			E_MA_EVENT.MA_MOVE:
				M_SetMode(RefCtrl.nMode);	
				M_SetStatus('Moving  ...');
				IF (RefStat.nMode = MA_MODE_ENG) THEN
					// Set nCyclesIdle to zero.
					// Needed to distinguish if the motor is about to move off or it completed the move.
					RefStat.nSkippedCycles	:= 0;
					M_NextMove();		// Set new position and move absolute
					SetState(E_MA_STATE.OP, E_MA_SUBSTATE.OP_MOVING);
				ELSE
					M_NextMove();
//					SetState(E_MA_STATE.OP, E_MA_SUBSTATE.OP_TRACKING);
					SetState(E_MA_STATE.OP, E_MA_SUBSTATE.OP_PRESETTING);
				END_IF
			E_MA_EVENT.START_TRACK:
				M_SetMode(RefCtrl.nMode);	
				// Set nCyclesIdle to zero.
				// Needed to distinguish if the motor is about to move off or it completed the move.
				RefStat.nSkippedCycles 	:= 0;	// Delayed action
				M_NextMoveAbs();
//				SetState(E_MA_STATE.OP, E_MA_SUBSTATE.OP_TRACKING);
				SetState(E_MA_STATE.OP, E_MA_SUBSTATE.OP_PRESETTING);
			E_MA_EVENT.PRESETDONE:
				// Preset is done, start tracking.
				SetState(E_MA_STATE.OP, E_MA_SUBSTATE.OP_TRACKING);
			E_MA_EVENT.TRACKEXIT:
				// Tracking is not good, it's more like presetting.
				SetState(E_MA_STATE.OP, E_MA_SUBSTATE.OP_PRESETTING);
		END_CASE
END_CASE
END_METHOD

{attribute 'TcRpcEnable':='1'}
METHOD RPC_Init : INT
VAR_INPUT
END_VAR

VAR 
	i: INT;
	bMotorMoving:	BOOL := FALSE;
END_VAR
// Log similar string in every derived FB
//M_LogEventGeneral('Initialising MA motors');

//
// Check if it is safe to operate motors.
//
IF NOT in_bSafe	THEN
	RPC_Init	:= M_SetRpcStatus(E_MA_RPC_ERROR.UNSAFE);
	RETURN;
END_IF


// It does all the verifications for the MOTOR device before
// triggering the Init event.

FOR i := 1 TO nNumAxes DO
	// RPC calls are not allowed in Local mode.
	// Fail on the first occurrence.
	IF ptrMotorStat[i]^.bLocal THEN
		RPC_Init	:= M_SetRpcStatus(E_MA_RPC_ERROR.LOCAL);
		RETURN;
	END_IF

	// If any of the motors is moving, RPC_Init() will fail.
	// However, the moving motor will be stopped, so next INIT will be OK.
	// We loop through all motors.
	IF	ptrMotorStat[i]^.nState = E_MOTOR_STATE.OP	AND  
		ptrMotorStat[i]^.nSubstate <> E_MOTOR_SUBSTATE.OP_STANDSTILL	THEN
		// There is a moving motor in the system.
		bMotorMoving	:= TRUE;
		// Stop the motor.
		// Send STOP command to the motors.
		ptrMotorCtrl[i]^.nCommand	:= E_MOTOR_COMMAND.STOP;
		ptrMotorCtrl[i]^.bExecute	:= TRUE;
		// RPC_Init() will fail !!!
		RPC_Init	:= M_SetRpcStatus(E_MA_RPC_ERROR.INIT_WHILE_MOVING);
	END_IF
END_FOR

IF bMotorMoving THEN
	// RPC_Init is already set to failure.
	RETURN;
ELSE
	// Proceed with INIT.
	RefCtrl.nCommand := E_MA_COMMAND.INIT;
	RefCtrl.bExecute := TRUE;
		
	// Call was successful
	RPC_Init	:= M_SetRpcStatus(E_MA_RPC_ERROR.OK);
END_IF
END_METHOD

METHOD SetAction
VAR_INPUT
	actionName:		STRING;
END_VAR

RefStat.sm.sActionDesc := actionName;
END_METHOD

METHOD SetEvent
VAR_INPUT
	nEventId:			DINT;
END_VAR

nEvent := nEventId;

CASE nEventId OF
	E_MA_EVENT.NONE:
		RefStat.sm.sEventDesc := '';
		RETURN;
		
	E_MA_EVENT.RESET:
		RefStat.sm.sEventDesc := 'CMD RESET';
		RETURN;
	
	E_MA_EVENT.INIT:
		RefStat.sm.sEventDesc := 'CMD INIT';
		RETURN;

	E_MA_EVENT.STOP:
		RefStat.sm.sEventDesc := 'CMD STOP';
		RETURN;

	E_MA_EVENT.ENABLE:
		RefStat.sm.sEventDesc := 'CMD ENABLE';
		RETURN;

	E_MA_EVENT.DISABLE:
		RefStat.sm.sEventDesc := 'CMD DISABLE';
		RETURN;
		
	E_MA_EVENT.MA_MOVE:
		RefStat.sm.sEventDesc := 'CMD MOVE';
		RETURN;
		
	E_MA_EVENT.START_TRACK:
		RefStat.sm.sEventDesc := 'CMD START_TRACK -> PRESETTING';
		RETURN;

	E_MA_EVENT.STOP_TRACK:
		RefStat.sm.sEventDesc := 'CMD STOP_TRACK';
		RETURN;
		
	E_MA_EVENT.PRESETDONE:
		RefStat.sm.sEventDesc := 'TRACKING';
		RETURN;
		
	E_MA_EVENT.TRACKEXIT:
		RefStat.sm.sEventDesc := 'TRACKING -> PRESETTING';
		RETURN;
		
	E_MA_EVENT.HWOK:
		RefStat.sm.sEventDesc := 'SIG HWOK';
		RETURN;

	E_MA_EVENT.ERRHW:
		RefStat.sm.sEventDesc := 'INT ERRHW';
		RETURN;
	
	E_MA_EVENT.UNSAFE:
		RefStat.sm.sEventDesc := 'EXT UNSAFE';
		RETURN;
	
END_CASE 

(* INTERNAL ERROR *)
RefStat.sm.sEventDesc := 'UNKNOWN EVENT';
END_METHOD

// Set the state and substate of the device
METHOD SetState : BOOL
VAR_INPUT
	in_nState:		INT;
	in_nSubstate:	INT;
END_VAR

(* 
	Update State Machine active state configuration.
*)

IF in_nState <> E_MA_STATE.NONE THEN
	RefStat.sm.nState	:= in_nState;
END_IF
IF in_nSubstate <> E_MA_SUBSTATE.NONE THEN
	RefStat.sm.nSubstate	:= in_nSubstate;
END_IF

(* Update active state configuration description *)

IF in_nState = E_MA_STATE.NOTOP THEN
	RefStat.sm.sState	:= 'NOT OP';
ELSIF in_nState = E_MA_STATE.OP THEN
	RefStat.sm.sState	:= 'OPERATIONAL';
END_IF

IF in_nSubstate = E_MA_SUBSTATE.NOTOP_NOTREADY THEN
	RefStat.sm.sSubstate	:= 'NOT READY';
ELSIF in_nSubstate = E_MA_SUBSTATE.NOTOP_INITIALISING THEN
	RefStat.sm.sSubstate	:= 'INITIALISING';
ELSIF in_nSubstate = E_MA_SUBSTATE.NOTOP_READY THEN
	RefStat.sm.sSubstate	:= 'READY';
ELSIF in_nSubstate = E_MA_SUBSTATE.NOTOP_ERROR THEN
	RefStat.sm.sSubstate	:= 'ERROR';
ELSIF in_nSubstate = E_MA_SUBSTATE.OP_DISABLING THEN
	RefStat.sm.sSubstate	:= 'DISABLING';
ELSIF in_nSubstate = E_MA_SUBSTATE.OP_MOVING THEN
	RefStat.sm.sSubstate	:= 'MOVING';
ELSIF in_nSubstate = E_MA_SUBSTATE.OP_STANDSTILL THEN
	RefStat.sm.sSubstate	:= 'STANDSTILL';
ELSIF in_nSubstate = E_MA_SUBSTATE.OP_TRACKING THEN
	RefStat.sm.sSubstate	:= 'TRACKING';
ELSIF in_nSubstate = E_MA_SUBSTATE.OP_PRESETTING THEN
	RefStat.sm.sSubstate	:= 'PRESETTING';
ELSIF in_nSubstate = E_MA_SUBSTATE.OP_STOPPING THEN
	RefStat.sm.sSubstate	:= 'STOPPING';
ELSIF in_nSubstate = E_MA_SUBSTATE.OP_ERROR THEN
	RefStat.sm.sSubstate	:= 'ERROR';
ELSE
	RefStat.sm.sSubstate	:= '';
END_IF
END_METHOD

METHOD User_ComputeNextPos : BOOL
VAR_INPUT
END_VAR
VAR
	i:	int;
END_VAR
// TODOUSER: Calculate next position for each axes based on the current mode.
IF RefStat.nMode = MA_MODE_ENG THEN
	FOR i := 1 TO nNumAxes DO
		;
	END_FOR
END_IF
END_METHOD

// Method for hard-coding of configuration parameters by the User.
METHOD User_Configure : BOOL
VAR_INPUT
END_VAR
VAR
	i:	INT;
END_VAR
//
// TODOUSER: Configure anything that is different from default configuration or
//           that has to take all motors into account.
//

//
// This is mandatory.
//
// Set the global timeouts to the longest ones. 
FOR i := 1 TO nNumAxes DO
	IF ptrMotorCfg[i]^.nTimeoutInit > RefCfg.timeout.nInitTimeout THEN
		RefCfg.timeout.nInitTimeout  := ptrMotorCfg[i]^.nTimeoutInit;
	END_IF
	IF ptrMotorCfg[i]^.nTimeoutMove > RefCfg.timeout.nMoveTimeout THEN
		RefCfg.timeout.nMoveTimeout  := ptrMotorCfg[i]^.nTimeoutMove;
	END_IF
END_FOR

//
// TODOUSER: Any other configuration
//
END_METHOD

// User Method executed on each cycle before processing events and states.
METHOD User_GetParams : BOOL
VAR_INPUT
END_VAR
VAR
	i:	INT;
END_VAR
//
// TODOUSER: Set anything that should be set on every cycle, if any.
//

// Example: Any settings that are mode dependant.
CASE RefCtrl.nMode OF
			MA_MODE_ENG:
			    ; 
END_CASE
END_METHOD

// User Method executed on each cycle after processing events and states.
METHOD User_SetParams : BOOL
VAR_INPUT
END_VAR
VAR
	i:		INT;
END_VAR
//
// Mandatory
//
// Set maximum positioning error
RefStat.lrPosError	:= M_GetMaxPosError();


// TODO Add code for handling individual axes, if any.
FOR i := 1 TO nNumAxes DO
	;
END_FOR
END_METHOD

END_FUNCTION_BLOCK

// ---- POUs/MultiAxis/FB_MA_DROT.TcPOU
FUNCTION_BLOCK FB_MA_DROT EXTENDS FB_MA_BASE
VAR_INPUT
	{attribute 'OPC.UA.DA' := '0'}
	sMotorName:			STRING	:= 'Motor';	(* Default Motor name *)
	{attribute 'OPC.UA.DA' := '0'}
	in_lrRotation: LREAL := 0; (* Rotation used for Sky mode *)
	{attribute 'OPC.UA.DA' := '0'}
	in_lrPupil: LREAL := 0; (* Pupil rotation for Elevation mode *)
	{attribute 'OPC.UA.DA' := '0'}
	in_lrParallactic: LREAL := 0; (* Parallactic angle *)
	{attribute 'OPC.UA.DA' := '0'}
	nNOVRAM_DevId:	UDINT	:= 0;		(* NOVRAM device ID - normally 4 *)
	{attribute 'OPC.UA.DA' := '0'}
	nNOVRAM_Offset:	UDINT	:= 0;		(* NOVRAM offset where motor configuration is stored *)
END_VAR
VAR_OUTPUT
END_VAR
VAR

	
	{attribute 'OPC.UA.DA' := '1'}
	cfg:				T_DROT_CFG;
	{attribute 'OPC.UA.DA' := '1'}
	ctrl:				T_DROT_CTRL;
	{attribute 'OPC.UA.DA' := '1'}
	stat:				T_DROT_STAT;
	
	{attribute 'OPC.UA.DA':='1'}
	motor:              FB_MOTOR;
	
END_VAR


// A MUST !!! Set references to real structures
RefCfg		REF=cfg;
RefCtrl		REF=ctrl;
RefStat		REF=stat;


motor(	sName 				:= sMotorName,	
		in_bSafe			:= in_bSafe,
		in_bDisableIfUnsafe	:= in_bDisableIfUnsafe,
		nNOVRAM_DevId 		:= nNOVRAM_DevId, 
		nNOVRAM_Offset 		:= nNOVRAM_Offset);

SUPER^(nNumAxes:=1, pMotor1:=ADR(motor));

METHOD M_LogCommand : BOOL
VAR
	cmd:	INT;
	mode:	INT;
	sLog:	STRING;
END_VAR
cmd		:= RefCtrl.nCommand;
mode	:= ctrl.nMode;

// Log DROT command.
// Set motor logging to FALSE when tracking,
// in order to reduce flooding of logs.
IF cmd = E_MA_COMMAND.RESET THEN
	pMotor1^.RPC_SetLog(TRUE);
	M_SetStatus('Resetting DROT device...');		
	M_LogEventGeneral('Resetting DROT device...');
ELSIF cmd = E_MA_COMMAND.ENABLE THEN
	pMotor1^.RPC_SetLog(TRUE);
	M_SetStatus('');		
	M_LogEventGeneral('Enabling DROT device...');
ELSIF cmd = E_MA_COMMAND.INIT THEN
	pMotor1^.RPC_SetLog(TRUE);
	M_SetStatus('Initialising DROT device...');		
	M_LogEventGeneral('Initialising DROT device...');
ELSIF cmd = E_MA_COMMAND.START_TRACK THEN
	pMotor1^.RPC_SetLog(FALSE);
	IF mode= E_DROT_MODE.ELEV THEN
		M_SetStatus('Tracking in ELEV mode');
		sLog	:= LREAL_TO_STRING(ctrl.lrPosang);
		sLog	:= CONCAT('Setting DROT to ELEVATION mode. Angle = ', sLog);
		M_LogEventGeneral(sLog);
	ELSIF mode= E_DROT_MODE.SKY THEN
		M_SetStatus('Tracking in SKY mode');
		sLog	:= LREAL_TO_STRING(ctrl.lrPosang);
		sLog	:= CONCAT('Setting DROT to SKY mode. Angle = ', sLog);
		M_LogEventGeneral(sLog);
	ELSIF mode= E_DROT_MODE.USER THEN
		M_SetStatus('Tracking in USER mode');
		sLog	:= LREAL_TO_STRING(ctrl.lrPosang);
		sLog	:= CONCAT('Setting DROT to USER mode. Angle = ', sLog);
		M_LogEventGeneral(sLog);
	END_IF
ELSIF cmd = E_MA_COMMAND.DISABLE THEN
	M_SetStatus('');		
	M_LogEventGeneral('Disabling DROT device...');
ELSIF cmd = E_MA_COMMAND.STOP THEN
	pMotor1^.RPC_SetLog(TRUE);
	M_LogEventGeneral('Stopping DROT device...');
ELSIF cmd = E_MA_COMMAND.STOP_TRACK THEN
	pMotor1^.RPC_SetLog(TRUE);
	IF mode= E_DROT_MODE.ENG THEN
		M_SetStatus('Moving to Engineering position ...');		
		sLog	:= LREAL_TO_STRING(stat.lrPos);
		sLog	:= CONCAT('Setting DROT to ENG mode. Angle = ', sLog);
		M_LogEventGeneral(sLog);
	ELSIF mode= E_DROT_MODE.STAT THEN
		M_SetStatus('Moving to STAT position ...');		
		sLog	:= LREAL_TO_STRING(stat.lrPos);
		sLog	:= CONCAT('Setting DROT to STAT mode. Angle = ', sLog);
		M_LogEventGeneral(sLog);
	END_IF
END_IF
END_METHOD

{attribute 'TcRpcEnable':='1'}
METHOD RPC_Disable : INT
VAR_INPUT
END_VAR

// It does all the verifications for the MOTOR device before
// triggering the Init event.

// RPC calls are not allowed in Local mode.
IF ptrMotorStat[1]^.bLocal THEN
	RPC_Disable	:= M_SetRpcStatus(E_MA_RPC_ERROR.LOCAL);
	RETURN;
END_IF

// Disable command is accepted only if device is in OP state.
IF ptrMotorStat[1]^.nState <> E_MOTOR_STATE.OP THEN
	RPC_Disable	:= M_SetRpcStatus(E_MA_RPC_ERROR.NOT_OP);
	RETURN;
ELSE
	// Set disable command
	RefCtrl.nCommand := E_MA_COMMAND.DISABLE;
	RefCtrl.bExecute := TRUE;
	
	// Call was successful
	RPC_Disable	:= M_SetRpcStatus(E_MA_RPC_ERROR.OK);
END_IF
END_METHOD

{attribute 'TcRpcEnable':='1'}
METHOD RPC_Enable : INT
VAR_INPUT
END_VAR

// It does all the verifications for the MOTOR device before
// triggering the Enable event.

//
// Check if it is safe to operate motors.
//
IF NOT in_bSafe	THEN
	RPC_Enable	:= M_SetRpcStatus(E_MA_RPC_ERROR.UNSAFE);
	RETURN;
END_IF



// RPC calls are not allowed in Local mode.
IF ptrMotorStat[1]^.bLocal THEN
	RPC_Enable	:= M_SetRpcStatus(E_MA_RPC_ERROR.LOCAL);
	RETURN;
END_IF

// Enable command is accepted only if device is in NOTOP_READY.
IF	ptrMotorStat[1]^.nSubstate <> E_MOTOR_SUBSTATE.NOTOP_READY		THEN
	RPC_Enable	:= M_SetRpcStatus(E_MA_RPC_ERROR.NOT_NOTOP_READY);
	RETURN;
ELSE
	// Set enable command
	RefCtrl.nCommand := E_MA_COMMAND.ENABLE;
	RefCtrl.bExecute := TRUE;
	
	// Call was successful
	RPC_Enable	:= M_SetRpcStatus(E_MA_RPC_ERROR.OK);
END_IF
END_METHOD

{attribute 'TcRpcEnable':='1'}
METHOD RPC_Init : INT
VAR_INPUT
END_VAR

VAR
END_VAR
M_LogEventGeneral('Initialising DROT motor...');

//
// Check if it is safe to operate motors.
//
IF NOT in_bSafe	THEN
	RPC_Init	:= M_SetRpcStatus(E_MA_RPC_ERROR.UNSAFE);
	RETURN;
END_IF


RPC_Init	:= SUPER^.RPC_Init();
END_METHOD

{attribute 'TcRpcEnable':='1'}
METHOD RPC_MoveAbs : INT
VAR_INPUT
	in_lrPos:	LREAL;
	in_lrVel:	LREAL;
END_VAR
//
// Check if it is safe to operate motors.
//
IF NOT in_bSafe	THEN
	RPC_MoveAbs	:= M_SetRpcStatus(E_MA_RPC_ERROR.UNSAFE);
	RETURN;
END_IF


// RPC calls are not allowed in Local mode.
IF motor.stat.bLocal THEN
	RPC_MoveAbs	:= M_SetRpcStatus(E_MA_RPC_ERROR.LOCAL);
	RETURN;
// Move Absolute command is accepted only in OP state.
ELSIF	motor.stat.nState <> E_MOTOR_STATE.OP	THEN
	RPC_MoveAbs	:= M_SetRpcStatus(E_MA_RPC_ERROR.NOT_OP);
	RETURN;
ELSIF	stat.sm.nState <> E_MA_STATE.OP	THEN
	RPC_MoveAbs	:= M_SetRpcStatus(E_MA_RPC_ERROR.NOT_OP);
	RETURN;
// Set velocity cannot be <=0.0.
ELSIF	in_lrVel <= 0.0	THEN
	RPC_MoveAbs	:= M_SetRpcStatus(E_MOTOR_RPC_ERROR.VEL_NEG);
	RETURN;
// Set velocity cannot be greater than MAX Velocity.
ELSIF	in_lrVel > motor.stat.axis.lrMaxVelocity	THEN
	RPC_MoveAbs	:= M_SetRpcStatus(E_MOTOR_RPC_ERROR.VEL_MAX);
	RETURN;
END_IF


SetState(E_MA_STATE.OP, E_MA_SUBSTATE.OP_MOVING);
// Set command
ctrl.nCommand 		:= E_MA_COMMAND.MA_MOVE;
ctrl.nMode          := E_DROT_MODE.ENG;
ctrl.lrTargetPos    := in_lrPos;
ctrl.lrTargetVel    := in_lrVel;
ctrl.bExecute 		:= TRUE;

// Call was successful
RPC_MoveAbs	:= M_SetRpcStatus(E_MA_RPC_ERROR.OK);
END_METHOD

{attribute 'TcRpcEnable':='1'}
METHOD RPC_MoveAngle : INT
VAR_INPUT
	in_lrAngle:	LREAL;
END_VAR
//
// Check if it is safe to operate motors.
//
IF NOT in_bSafe	THEN
	RPC_MoveAngle	:= M_SetRpcStatus(E_MA_RPC_ERROR.UNSAFE);
	RETURN;
END_IF



// RPC calls are not allowed in Local mode.
IF motor.stat.bLocal THEN
	RPC_MoveAngle	:= M_SetRpcStatus(E_MA_RPC_ERROR.LOCAL);
	RETURN;
// Move Absolute command is accepted only in OP state.
ELSIF	motor.stat.nState <> E_MOTOR_STATE.OP	THEN
	RPC_MoveAngle	:= M_SetRpcStatus(E_MA_RPC_ERROR.NOT_OP);
	RETURN;
ELSIF	stat.sm.nState <> E_MA_STATE.OP	THEN
	RPC_MoveAngle	:= M_SetRpcStatus(E_MA_RPC_ERROR.NOT_OP);
	RETURN;
END_IF


SetState(E_MA_STATE.OP, E_MA_SUBSTATE.OP_MOVING);
// Set command
ctrl.lrPosang 	:= in_lrAngle;
ctrl.nMode		:= E_DROT_MODE.STAT;
ctrl.nCommand	:= E_MA_COMMAND.STOP_TRACK;
ctrl.bExecute	:= TRUE;

// Call was successful
RPC_MoveAngle	:= M_SetRpcStatus(E_MA_RPC_ERROR.OK);
END_METHOD

{attribute 'TcRpcEnable':='1'}
METHOD RPC_MoveRel : INT
VAR_INPUT
	in_lrPos:	LREAL;
	in_lrVel:	LREAL;
END_VAR
//
// Check if it is safe to operate motors.
//
IF NOT in_bSafe	THEN
	RPC_MoveRel	:= M_SetRpcStatus(E_MA_RPC_ERROR.UNSAFE);
	RETURN;
END_IF


// RPC calls are not allowed in Local mode.
IF motor.stat.bLocal THEN
	RPC_MoveRel	:= M_SetRpcStatus(E_MA_RPC_ERROR.LOCAL);
	RETURN;
// Move Absolute command is accepted only in OP state.
ELSIF	motor.stat.nState <> E_MOTOR_STATE.OP	THEN
	RPC_MoveRel	:= M_SetRpcStatus(E_MA_RPC_ERROR.NOT_OP);
	RETURN;
ELSIF	stat.sm.nState <> E_MA_STATE.OP	THEN
	RPC_MoveRel	:= M_SetRpcStatus(E_MA_RPC_ERROR.NOT_OP);
	RETURN;
// Set velocity cannot be <=0.0.
ELSIF	in_lrVel <= 0.0	THEN
	RPC_MoveRel	:= M_SetRpcStatus(E_MOTOR_RPC_ERROR.VEL_NEG);
	RETURN;
// Set velocity cannot be greater than MAX Velocity.
ELSIF	in_lrVel > motor.stat.axis.lrMaxVelocity	THEN
	RPC_MoveRel	:= M_SetRpcStatus(E_MOTOR_RPC_ERROR.VEL_MAX);
	RETURN;
END_IF


SetState(E_MA_STATE.OP, E_MA_SUBSTATE.OP_MOVING);
// Set command
ctrl.nCommand 		:= E_MA_COMMAND.MA_MOVE;
ctrl.nMode          := E_DROT_MODE.ENG;
ctrl.lrTargetPos    := motor.stat.lrPosActual + in_lrPos;
ctrl.lrTargetVel    := in_lrVel;
ctrl.bExecute 		:= TRUE;

// Call was successful
RPC_MoveRel	:= M_SetRpcStatus(E_MA_RPC_ERROR.OK);
END_METHOD

{attribute 'TcRpcEnable':='1'}
METHOD RPC_MoveVel : INT
VAR_INPUT
	in_lrVel:	LREAL;
END_VAR
VAR
	dir:	DINT;
END_VAR
//
// Check if it is safe to operate motors.
//
IF NOT in_bSafe	THEN
	RPC_MoveVel	:= M_SetRpcStatus(E_MA_RPC_ERROR.UNSAFE);
	RETURN;
END_IF


IF	stat.sm.nState <> E_MA_STATE.OP	THEN
	RPC_MoveVel	:= M_SetRpcStatus(E_MA_RPC_ERROR.NOT_OP);
	RETURN;
ELSIF	in_lrVel = 0.0	THEN
// Set velocity cannot be 0.0.
	RPC_MoveVel	:= M_SetRpcStatus(E_MOTOR_RPC_ERROR.VEL_ZERO);
	RETURN;
END_IF

// Check velocity against Vel_max.
// Note: Negative velocity is accepted.
// Check if Velocity is too high.
IF ABS(in_lrVel) > ptrMotorStat[1]^.axis.lrMaxVelocity THEN
	RPC_MoveVel	:= M_SetRpcStatus(E_MOTOR_RPC_ERROR.VEL_MAX);
	RETURN;
END_IF


// Update State and Status
SetState(E_MA_STATE.OP, E_MA_SUBSTATE.OP_MOVING);
M_SetStatus('Moving in Velocity mode...');
ctrl.nMode	:= E_ADC_MODE.ENG;

// Set the direction of movement.
IF in_lrVel > 0.0	THEN
	dir	:= MC_Positive_Direction;
ELSE
	dir	:= MC_Negative_Direction;
END_IF

// This will command all the motors and restart the timer.
ActionMoveVelExecute(vel:=ABS(in_lrVel), dir:=dir);

// Call was successful
RPC_MoveVel	:= M_SetRpcStatus(E_MA_RPC_ERROR.OK);
END_METHOD

{attribute 'TcRpcEnable':='1'}
METHOD RPC_Reset : INT
VAR_INPUT
END_VAR

// RPC calls are not allowed in Local mode.
IF ptrMotorStat[1]^.bLocal THEN
	RPC_Reset	:= M_SetRpcStatus(E_MA_RPC_ERROR.LOCAL);
	RETURN;
END_IF

ctrl.nCommand := E_MA_COMMAND.RESET;
ctrl.bExecute := TRUE;

// Call was successful
RPC_Reset	:= M_SetRpcStatus(E_MA_RPC_ERROR.OK);
END_METHOD

{attribute 'TcRpcEnable':='1'}
METHOD RPC_StartTrack : INT
VAR_INPUT
	in_mode:	 INT := 2;
	in_angle:    LREAL := 0.0;
END_VAR
//
// Check if it is safe to operate motors.
//
IF NOT in_bSafe	THEN
	RPC_StartTrack	:= M_SetRpcStatus(E_MA_RPC_ERROR.UNSAFE);
	RETURN;
END_IF



// RPC calls are not allowed in Local mode.
IF ptrMotorStat[1]^.bLocal THEN
	RPC_StartTrack	:= M_SetRpcStatus(E_MA_RPC_ERROR.LOCAL);
	RETURN;
// Move Absolute command is accepted only in OP state.
ELSIF	ptrMotorStat[1]^.nState <> E_MOTOR_STATE.OP	THEN
	RPC_StartTrack	:= M_SetRpcStatus(E_MA_RPC_ERROR.NOT_OP);
	RETURN;
END_IF

// Set command
ctrl.lrPosang := in_angle;
ctrl.nMode:= in_mode;
ctrl.nCommand:=E_MA_COMMAND.START_TRACK;
ctrl.lrOffset := 0.0;
stat.lrTotalOffset := 0.0;
ctrl.bExecute:=(TRUE);

// Call was successful
RPC_StartTrack	:= M_SetRpcStatus(E_MA_RPC_ERROR.OK);
END_METHOD

{attribute 'TcRpcEnable':='1'}
METHOD RPC_Stop : INT
VAR_INPUT
END_VAR

// RPC calls are not allowed in Local mode.
IF ptrMotorStat[1]^.bLocal THEN
	RPC_Stop	:= M_SetRpcStatus(E_MA_RPC_ERROR.LOCAL);
	RETURN;
END_IF

ctrl.nCommand := E_MA_COMMAND.STOP;
ctrl.bExecute := TRUE;

RPC_Stop	:= M_SetRpcStatus(E_MA_RPC_ERROR.OK);
END_METHOD

{attribute 'TcRpcEnable':='1'}
METHOD RPC_StopTrack : INT
VAR_INPUT
END_VAR
VAR
	sLog:	STRING;
END_VAR
IF (RefStat.nMode >= E_DROT_MODE.SKY) THEN
	// RPC calls are not allowed in Local mode.
	IF ptrMotorStat[1]^.bLocal THEN
		RPC_StopTrack	:= M_SetRpcStatus(E_MA_RPC_ERROR.LOCAL);
		RETURN;
	END_IF

	sLog	:= LREAL_TO_STRING(stat.lrPos);
	sLog	:= CONCAT('Stopping Tracking. Angle = ', sLog);
	M_LogEventGeneral(sLog);

	RefCtrl.nMode           :=  E_DROT_MODE.STAT;
	// Set command
	RefCtrl.nCommand 		:= E_MA_COMMAND.STOP_TRACK;
	RefCtrl.bExecute 		:= TRUE;
END_IF

// Call was successful
RPC_StopTrack	:= M_SetRpcStatus(E_MA_RPC_ERROR.OK);
END_METHOD

{attribute 'TcRpcEnable':='1'}
METHOD RPC_TrackOffset : INT
VAR_INPUT
	in_lrOffset:	LREAL;
END_VAR
//
// Check if it is safe to operate motors.
//
IF NOT in_bSafe	THEN
	RPC_TrackOffset	:= M_SetRpcStatus(E_MA_RPC_ERROR.UNSAFE);
	RETURN;
END_IF


// RPC calls are not allowed in Local mode.
IF motor.stat.bLocal THEN
	RPC_TrackOffset	:= M_SetRpcStatus(E_MA_RPC_ERROR.LOCAL);
	RETURN;
// Move Absolute command is accepted only in OP state.
ELSIF	motor.stat.nState <> E_MOTOR_STATE.OP	THEN
	RPC_TrackOffset	:= M_SetRpcStatus(E_MA_RPC_ERROR.NOT_OP);
	RETURN;
ELSIF	(stat.nMode <= E_DROT_MODE.STAT) THEN
	RPC_TrackOffset	:= M_SetRpcStatus(E_MA_RPC_ERROR.NOT_TRACKING);
	RETURN;
END_IF

// Update offset
ctrl.lrOffset    := in_lrOffset;

// Call was successful
RPC_TrackOffset	:= M_SetRpcStatus(E_MA_RPC_ERROR.OK);
END_METHOD

METHOD User_ComputeNextPos : BOOL
VAR_INPUT
END_VAR
VAR
	fieldRotation: LREAL;
	modeAngle:     LREAL;
	pos:           LREAL := 0.0 ;
	posang:        LREAL;
END_VAR
// Handle various derotator modes
CASE RefCtrl.nMode OF
			E_DROT_MODE.STAT:
			    pos := cfg.lrStatRef + cfg.nDirSign * (ctrl.lrPosang)/2.0;
				stat.lrAngleOnSky := 0.0;
				stat.lrModeAngle := pos;
				ptrMotorCtrl[1]^.lrVelocity := ptrMotorCfg[1]^.lrDefaultVelocity;
			E_DROT_MODE.SKY:
				stat.lrTotalOffset := stat.lrTotalOffset + ctrl.lrOffset;
				ctrl.lrOffset := 0.0;
				fieldRotation := ctrl.lrRotation;
				pos := cfg.lrSkyRef + (cfg.nDirSign * ((ctrl.lrPosang - fieldRotation)/2)) + stat.lrTotalOffset ;
				stat.lrAngleOnSky := ctrl.lrPosang;
				stat.lrModeAngle := stat.lrAngleOnSky;
				ptrMotorCtrl[1]^.lrVelocity := ptrMotorCfg[1]^.lrDefaultVelocity;
			E_DROT_MODE.ELEV:
				stat.lrTotalOffset := stat.lrTotalOffset + ctrl.lrOffset;
				ctrl.lrOffset := 0.0;
				pos := cfg.lrElevRef + ((cfg.nFocusSign * cfg.nDirSign * (ctrl.lrPupil)) /2.0) + stat.lrTotalOffset;
				stat.lrAngleOnSky := ctrl.lrParallactic;
				stat.lrModeAngle := stat.lrAngleOnSky;
				ptrMotorCtrl[1]^.lrVelocity := ptrMotorCfg[1]^.lrDefaultVelocity;
			E_DROT_MODE.USER:
				//modeAngle := (parUser[1] * ctrl.lrPosang +
				//	          parUser[2] * i_trk_data.alt_deg +
				//			  parUser[3] * i_trk_data.pa_deg );
				//pos := cfg.lrUserRef + cfg.nDirSign * modeAngle;
				//stat.lrAngleOnSky := 0.0;
				//stat.lrModeAngle  := modeAngle;
			E_DROT_MODE.ENG:
				pos := ctrl.lrTargetPos;
		        ptrMotorCtrl[1]^.lrVelocity := ctrl.lrTargetVel;		
		        M_SetStatus('Moving to Engineering position ...');
END_CASE

// assign new TARGET position
ptrMotorCtrl[1]^.lrPosition := pos;
stat.lrPos := pos;	// Used in the DROT GUI as 'Target'
END_METHOD

// Method for hard-coding of configuration parameters by the User.
METHOD User_Configure : BOOL
VAR_INPUT
END_VAR
VAR
	i:	INT;
END_VAR
SUPER^.User_Configure();	// Mandatory!

//
// TODOUSER: Configure anything that is different from default configuration.
//
// Examples:
//

//
// Individual Motor configuration
ptrMotorCfg[1]^.nAxisType	        := E_MOTOR_AXIS_TYPE.CIRCULAR_OPTIMISED;
ptrMotorCfg[1]^.lrDefaultVelocity	:= 3.0;	// Set default velocity to 10 deg/sec


// Multi-axis system configuration
ctrl.lrPosang	    :=  0.0;	// Position angle for OFF mode, i.e. HOME position
ctrl.lrTargetPos	:=  0.0;	
ctrl.lrTargetVel	:= 3.0;	// Velocity for ENG mode
END_METHOD

// User Method executed on each cycle before processing events and states.
METHOD User_GetParams : BOOL
VAR_INPUT
END_VAR
VAR
	i:	INT;
END_VAR


SUPER^.User_GetParams();
END_METHOD

// User Method executed on each cycle after processing events and states.
METHOD User_SetParams : BOOL
VAR_INPUT
END_VAR
VAR
	i:		INT;
END_VAR
//
// Mandatory
//
SUPER^.User_SetParams();

// Set maximum positioning error
stat.lrPosError		:= M_GetMaxPosError();

// Check if we are tracking or still presetting.
// Tracking is OK if the positioning error is less than the threshold (bTrackingOK).
// Once device is tracking, it should go back to presetting if the error is greater
// than twice the threshold  (bTrackingBAD).
IF	ctrl.nMode = E_DROT_MODE.ELEV OR  
	ctrl.nMode = E_DROT_MODE.SKY  OR  
	ctrl.nMode = E_DROT_MODE.USER	THEN
	stat.bTrackingOK	:= SEL (stat.lrPosError <= cfg.lrTrkThreshold, FALSE, TRUE);
	stat.bTrackingBAD	:= SEL (stat.lrPosError > 2.0 * cfg.lrTrkThreshold, FALSE, TRUE);
	ctrl.lrRotation := in_lrRotation;
	ctrl.lrPupil := in_lrPupil;
	stat.lrRotation := in_lrRotation;
	stat.lrPupil := in_lrPupil;
	ctrl.lrParallactic := in_lrParallactic;
ELSE
	stat.bTrackingOK	:= FALSE;
	stat.bTrackingBAD	:= FALSE;
END_IF
END_METHOD

END_FUNCTION_BLOCK

// ---- POUs/Functions/F_DCTIME64_TO_ULINT.TcPOU
FUNCTION F_DCTIME64_TO_ULINT : ULINT
VAR_INPUT
	in:		T_DCTIME64;
END_VAR
VAR
	out:	ULINT;
END_VAR

memcpy (ADR(out), ADR(in), SIZEOF(in));
F_DCTIME64_TO_ULINT	:= out;

END_FUNCTION

// ---- POUs/Functions/F_MOD.TcPOU
FUNCTION F_MOD : LREAL
VAR_INPUT
	A:	LREAL;
	B:	LREAL;
END_VAR
VAR
END_VAR

(*
#define vltMOD(A,B) 
((B)!=0.0?
	((A)*(B)>0.0?
		(A)-(B)*floor((A)/(B))
	else
		:(A)+(B)*floor(-(A)/(B)))
else
	:(A))
*)
IF B = 0.0 THEN
	F_MOD	:= A;
ELSE
	IF A * B >= 0.0 THEN
		F_MOD	:= A - B * TRUNC_INT(A / B);
	ELSE
		F_MOD	:= A + B * TRUNC_INT(-A / B);
	END_IF
END_IF

END_FUNCTION

// ---- POUs/Functions/F_RAD2DMS_STRING.TcPOU
FUNCTION F_RAD2DMS_STRING : STRING
VAR_INPUT
	dec:	LREAL;
END_VAR
VAR
	value:		LREAL;
	degrees:	INT;
	minutes:	INT;
	seconds:	LREAL;
	
	sign:	int := 1;
	result:	STRING := '';
	
	fbFormat   : FB_FormatString;
END_VAR

IF dec < 0.0 THEN
	sign	:= -1;
	dec		:= -dec;
END_IF

value := dec * GCL.C_RAD2DEG; 	// rad to hours


degrees	:= TRUNC_INT(value);
minutes := TRUNC_INT((value - degrees)*60.0);
seconds := (value - degrees - minutes/60.0)*3600.0;

// We the calculation so far the value of 14.999999999 will result
// in 14:59:60.
// We want to correct it to 15:00:00.
IF seconds > 59.999 THEN
	seconds	:= 0.0;
	minutes	:= minutes + 1;
	IF minutes = 60 THEN
		minutes	:= 0;
		degrees	:= degrees + 1;
	END_IF
// Seconds should never be < 0.0. However, it happens due to rounding
// and the value could be ~ -1.0 e-12.
// Set it to zero in that case.
ELSIF seconds < 0.0 THEN
	seconds := 0.0;
END_IF

degrees	:= degrees * sign;	// put back the sign

// format a string like "+07:01:02.123"
fbFormat( sFormat  := '%+.3d:%.2d:%06.3f', 
					arg1 := F_INT(degrees), 
					arg2 := F_INT(minutes), 
					arg3 := F_LREAL(seconds),
					sOut => result);
					
F_RAD2DMS_STRING	:= result;

END_FUNCTION

// ---- POUs/Functions/F_RAD2HMS_STRING.TcPOU
FUNCTION F_RAD2HMS_STRING : STRING
VAR_INPUT
	hh:	LREAL;
END_VAR
VAR
	value:		LREAL;
	hours:		INT;
	minutes:	INT;
	seconds:	LREAL;
	
	sign:	int := 1;
	result:	STRING := '';
	
	fbFormat   : FB_FormatString;
END_VAR

IF hh < 0.0 THEN
	sign	:= -1;
	hh		:= -hh;
END_IF

value := hh / GCL.C_2PI * 24.0; 	// rad to hours


hours	:= TRUNC_INT(value);
minutes := TRUNC_INT((value - hours)*60.0);
seconds := (value - hours - minutes/60.0)*3600.0;

// We the calculation so far the value of 14.999999999 will result
// in 14:59:60.
// We want to correct it to 15:00:00.
IF seconds > 59.999 THEN
	seconds	:= 0.0;
	minutes	:= minutes + 1;
	IF minutes = 60 THEN
		minutes	:= 0;
		hours	:= hours + 1;
	END_IF
// Seconds should never be < 0.0. However, it happens due to rounding
// and the value could be ~ -1.0 e-12.
// Set it to zero in that case.
ELSIF seconds < 0.0 THEN
	seconds := 0.0;
END_IF

hours	:= hours * sign;	// put back the sign

// format a string like "+07:01:02.123"
fbFormat( sFormat  := '%+.2d:%.2d:%06.3f', 
					arg1 := F_INT(hours), 
					arg2 := F_INT(minutes), 
					arg3 := F_LREAL(seconds),
					sOut => result);
					
F_RAD2HMS_STRING	:= result;

END_FUNCTION

// ---- POUs/Functions/F_timeGetAbsoluteDcTime.TcPOU
(*
 *****************************************************************************
 * timeGetAbsoluteDcTime: Adjust DC time based on the external time signal
 *
 *  IN   ptptime    : External time signal
 *  IN   leapSecond : Leap Second 
 *  OUT  dcTIME     : Adjusted TwinCAT DC time
 ***************************************************************************** 
 *)
FUNCTION F_timeGetAbsoluteDcTime : BOOL
VAR_INPUT
	ptptime:			T_ASTRO_EL6688_DATA;
	nLeapSecond:		DINT;
	DcToExtTimeOffset:	LINT;
END_VAR
VAR_IN_OUT
	dcTime:   ULINT;
END_VAR
VAR
	val:		LINT	:= 0;
	diff:		LINT	:= 0;
	one_sec:	LINT	:= 1000000000;
END_VAR

(*
HRESULT timeGetAbsoluteDcTime(PTPTime ptptime, INT leapSecond, LONGLONG *dcTime)
{
	HRESULT hr = S_OK; 
	LONGLONG val = 0;
	LONGLONG diff = 0;
	LONGLONG ONE_SEC = 1000000000;
	
	// Check if external time signal is connected
	if (ptptime.not_connected)
		return S_FALSE;

	// If both variables are null means most probably they are not mapped.
	if (ptptime.internal == 0 || ptptime.external == 0)
		return S_FALSE;

	diff = (ptptime.internal - ptptime.external) + (ONE_SEC * leapSecond) + ptptime.dcTcOffset;
	*dcTime -=  diff;
	return hr;
}*)

// Check if external time signal is connected
IF ptptime.External_device_not_connected THEN
	F_timeGetAbsoluteDcTime := FALSE;
END_IF

// If both variables are null means most probably they are not mapped.
// TODO: Is it OR or AND ?
IF ptptime.Internal_time_stamp = 0  OR  ptptime.External_time_stamp = 0 THEN
	F_timeGetAbsoluteDcTime := FALSE;
END_IF

diff := (ULINT_TO_LINT(ptptime.Internal_time_stamp) - ULINT_TO_LINT(ptptime.External_time_stamp)) + 
		(one_sec * nLeapSecond) + DcToExtTimeOffset;

dcTime	:= dcTime - LINT_TO_ULINT(diff);

F_timeGetAbsoluteDcTime := TRUE;

END_FUNCTION

// ---- POUs/Functions/F_timeGetDcTime.TcPOU
(*
 *****************************************************************************
 * timeGetDcTime: Get TwinCAT DC time from UTC time
 *
 *  IN   vltUTC: UTC time 
 *  OUT  dcTIME: TwinCAT DC time
 ***************************************************************************** 
 *)
FUNCTION F_timeGetDcTime : ULINT
VAR_INPUT
	ut:	T_TIMEVAL;
END_VAR
VAR
	val:   	ULINT := 0;
END_VAR

(*
HRESULT timeGetDcTime(vltTIMEVAL vltUTC, LONGLONG *dcTime)
{
	HRESULT hr = S_OK; 
	LONGLONG val = 0;
	val = vltUTC.tv_sec * 1000000000;
	val -= OFFSET_UNIX;
	*dcTime = val + vltUTC.tv_usec * 1000;
	return hr;
}
*)
val	:= ut.tv_sec * 1000000000;
val := val - DINT_TO_ULINT(GCL.C_OFFSET_UNIX);

F_timeGetDcTime	:= val + DINT_TO_ULINT(ut.tv_usec) * 1000;

END_FUNCTION

// ---- POUs/Misc/FB_DIGITAL_SIGNAL_FILTER.TcPOU
// 
// Filtering of digital signal in order to remove glitches.
// It returns the dominant signal level (FALSE or TRUE) during
// the period of in_nPeriod_ms.
// It is a moving window. Therefore the output is 
// recalculated on every PLC cycle.
//
// Variable mapping:
//   i_bSig - Linked to the physical input signal coming from the switch.
//   q_bSig - Filtered output signal to be linked to motor switch var.
//
// Usage:
// 	df:	FB_DIGITAL_SIGNAL_FILTER;
//  df(in_nPeriod_ms:=nPeriod_ms);
//
FUNCTION_BLOCK FB_DIGITAL_SIGNAL_FILTER
VAR_INPUT
	// Sampling period [ms].
	// Resulting delay in signal change = MAX((period/2),in_nConseqToggle) + 1 cycle.
	// Switch detection error = (motor travel during (in_nPeriod_ms/2 + 1 cycle)).
	//
	// Example:
	//    PLC cycle = 1 ms
	//    in_nPeriod_ms = 7 ms  ==> nTotal = 7 (7 samples to process).
	//    in_nConseqToggle = 3 samples
	//    delay = MAX((7/2,3) + 1 = 3 + 1 = 4 PLC cycles
	//    The signal level that appeares >=3 times out of 5 samples,
	//    determines the resulting level TRUE/FALSE.
	//    Needed accuracy in switch detection = 0.6 um = 0.0006 mm.
	//    V = D / T  = 0.0006 / (4/1000) 
	//      = 0.0006 / (4/1000) = 0.0006 / 0.004 = 0.15 mm/sec
	//
	//    Conclusion: 
	//       The fine motor velocity for switch detection should be <= 0.15 mm/sec.
	//
	in_nPeriod_ms:		UINT := 5;	
	// Minimum consequtive toggles to toggle the filtered output.
	in_nConseqToggle:	UINT := 2;	
END_VAR
VAR
	//
	// Signals to map.
	//
	// Physical input signal that we want to process/filter.
	i_bSig     AT %I*: BOOL;
	// Generated filtered output signal.
	// The input signal, e.g., motor limit switch, should
	// be mapped to this signal instead of i_bSig.
	q_bSig     AT %Q*: BOOL;
	
	fbGetCurTaskIdx:	GETCURTASKINDEX;
	nCycleTime:			UDINT;	// Cycle time in microsec.

	nToggles: 		UINT := 0;
	nConseqToggles: UINT := 0;
	nTotal:			UINT;	// Total number of samples.
	// Number of consequtive same readings to swap the output.
	nToggleLimit: 	UINT := 1;	
	
	bReady:			BOOL;	// If TRUE, the FB is configured.
	
END_VAR

// Find out the total number of samples, i.e., PLC cycles.
IF NOT bReady	THEN

	// Get cycle time in microsec.
	// CycleTime in _TaskInfo is given in 100 ns. 1 us = 1000 ns
	fbGetCurTaskIdx();
	nCycleTime	:=  (TwinCAT_SystemInfoVarList._TaskInfo[fbGetCurTaskIdx.index].CycleTime)/10;

	// Get total number of samples to process
	nTotal	:= UDINT_TO_UINT(1000 * in_nPeriod_ms / nCycleTime);

	// There should be at least three samples
	nTotal	:= MAX(nTotal, 3);
	// Number of samples should be an odd number, i.e., 3, 5, 7, etc.
	IF nTotal MOD 2 = 0	THEN
		nTotal	:= nTotal + 1;
	END_IF

	// The number of consecutive cycles with opposite value
	// before swapping the output.
	nToggleLimit	:= nTotal / 2 + 1;

	bReady := TRUE;
	
	RETURN;
END_IF


//
// System is configured, i.e., ready to run.
//

//
// Check if the input signal is the same as the filtered output.
//
IF i_bSig <> q_bSig THEN
	IF nToggles > 1  AND  nConseqToggles = 0	THEN
		// The previous non-toggle lasted only one sample,
		// This was a glitch.
		// Discard it by incrementing toggles by 2 
		// {this one plus the previous one)
		nToggles 		:= nToggles + 2;
	ELSE
		nToggles 		:= nToggles + 1;
	END_IF
	
	// Increment the number of consequtive toggles.
	nConseqToggles	:= nConseqToggles + 1;
	// At least in_nConseqToggle consequtive toggle readings
	// needed to toggle the filtered signal.
	IF nToggles >= nToggleLimit  AND  nConseqToggles >= in_nConseqToggle 	THEN
		// Toggle output
		q_bSig 			:= NOT q_bSig;
		nToggles		:= 0;
		nConseqToggles	:= 0;	
	END_IF
ELSE
	IF nToggles = 1  AND  nConseqToggles = 1	THEN
		// There was a toggle in the previous sample,
		// but now there is no toggle.
		// This was a glitch.
		nToggles		:= 0;	
	ELSE
		// Decrement the number of toggles.
		IF nToggles > 1	THEN
			nToggles := nToggles - 1;
		ELSE	
			nToggles := 0;
		END_IF
	END_IF
	
	// Reset the counter for consequtive toggles.
	nConseqToggles	:= 0;	
END_IF

END_FUNCTION_BLOCK

// ---- POUs/MultiAxis/FB_TRK_BASE.TcPOU
FUNCTION_BLOCK FB_TRK_BASE EXTENDS FB_MA_BASE
VAR_INPUT
END_VAR
VAR_OUTPUT
END_VAR
VAR
	{attribute 'OPC.UA.DA' := '0'}
	TrkCfg:		        REFERENCE TO T_TRK_CFG;	    // Reference to Config parameters
	{attribute 'OPC.UA.DA' := '0'}
	TrkCtrl:		    REFERENCE TO T_TRK_CTRL;	// Reference to Control parameters
	{attribute 'OPC.UA.DA' := '0'}
	TrkStat:		    REFERENCE TO T_TRK_STAT;	// Reference to Status parameters
	
    // Tracking data structure (TrackingData) is defined in C++ module
	{attribute 'OPC.UA.DA' := '0'}
	i_trk_data          AT %I*: PointingKernelPositions;
	
	{attribute 'OPC.UA.DA' := '0'}
	i_ccs_data          AT %I*: CcsData;
	
	
	
END_VAR



SUPER^();

// Method for hard-coding of configuration parameters by the User.
METHOD User_Configure : BOOL
VAR_INPUT
END_VAR
VAR
	i:	INT;
END_VAR
SUPER^.User_Configure();	// Mandatory!
END_METHOD

// User Method executed on each cycle before processing events and states.
METHOD User_GetParams : BOOL
VAR_INPUT
END_VAR
VAR
	i:	INT;
END_VAR

// Assign output variables according input configuration and control.
END_METHOD

// User Method executed on each cycle after processing events and states.
METHOD User_SetParams : BOOL
VAR_INPUT
END_VAR
VAR
	i:		INT;
END_VAR

memcpy(ADR(TrkCfg.site), ADR(i_ccs_data.site), SIZEOF(TrkCfg.site));
memcpy(ADR(TrkCtrl.environment), ADR(i_ccs_data.environment), SIZEOF(TrkCtrl.environment));
memcpy(ADR(TrkStat.data), ADR(i_trk_data), SIZEOF(TrkStat.data));
memcpy(ADR(TrkStat.data_deg), ADR(i_trk_data), SIZEOF(TrkStat.data_deg));
TrkStat.data_deg.target_observed_altaz[0] := RAD_TO_DEG(TrkStat.data.target_observed_altaz[0]);
TrkStat.data_deg.target_observed_altaz[1] := RAD_TO_DEG(TrkStat.data.target_observed_altaz[1]);
TrkStat.data_deg.parallactic_angle := RAD_TO_DEG(TrkStat.data.parallactic_angle);
TrkStat.data_deg.north_angle := RAD_TO_DEG(TrkStat.data.north_angle);
TrkStat.data_deg.pupil_angle := RAD_TO_DEG(TrkStat.data.pupil_angle);
TrkStat.apparent.alpha := F_astroRad2Hms(i_trk_data.radec_at_altaz_at_requested_xy[0]);
TrkStat.apparent.delta := F_astroRad2Dms(i_trk_data.radec_at_altaz_at_requested_xy[1]);
END_METHOD

END_FUNCTION_BLOCK

// ---- GlobalTextList.TcGTLO
TEXTLIST GlobalTextList
  830 = '\nNOT OP'
  834 = ' \n     OPERATIONAL'
  150 = ' 0 - END [0] [0] (e.g. "END,0,0")'
  151 = ' 1 - Find Index Switch [fast Vel] [slow Vel] (e.g. "FIND_INDEX,10.0,0.5")'
  152 = ' 2 - Find REF Switch Lower Edge [fast Vel] [slow Vel] (e.g. "FIND_REF_LE,8,0.1")'
  153 = ' 3 - Find REF Switch Upper Edge [fast Vel] [slow Vel] (e.g. "FIND_REF_UE,8.5,1")'
  154 = ' 4 - Find Lower HW Limit [fast Vel] [slow Vel] (e.g. "FIND_LHW,5.0,0.2")'
  155 = ' 5 - Find Upper HW Limit [fast Vel] [slow Vel] (e.g. "FIND_UHW,5.0,0.2")'
  160 = ' 6 - Delay [ms] [0] (e.g. "DELAY,3000,0")'
  156 = ' 7 - Move Absolute [vel] [pos] (e.g. "MOVE_ABS,25.0,360.0")'
  157 = ' 8 - Move Relative [vel] [pos] (e.g. "MOVE_REL,25.0,60.0")'
  158 = ' 9 - Calibrate Absolute [pos] [0] (e.g. "CALIB_ABS,180.0,0")'
  923 = '%.0f'
  24 = '%.1f'
  14 = '%.2f'
  3159 = '%.2lf'
  508 = '%.3f'
  321 = '%.4f'
  895 = '%.5f'
  343 = '%.6f'
  860 = '%d'
  11 = '%s'
  1022 = "'Motor.library version'"
  346 = '1'
  710 = '10'
  159 = '10 - Calibrate Relative [pos] [0] (e.g. "CALIB_REL,5.25,0")'
  161 = '11 - Calibrate on Switch [pos] [0.0] (e.g. "CALIB_SWITCH,180.0,0")'
  347 = '2'
  348 = '3'
  349 = '4'
  350 = '5'
  351 = '6'
  352 = '7'
  353 = '8'
  703 = '9'
  844 = 'ABORTING'
  753 = 'Absolute position used by "MOVE ABS"'
  519 = 'Action'
  149 = 'Action Legend:'
  178 = 'Active Low'
  1331 = 'Actual'
  23 = 'Actual Pos:'
  1074 = 'Actual time'
  849 = 'Actual Vel:'
  1657 = 'ADA :'
  1649 = 'Adapter position [deg]'
  9 = 'ADC control'
  1201 = 'ADC Control'
  852 = 'ADC Status'
  1625 = 'ADC1'
  1632 = 'ADC1 ENG position angle [deg]'
  1717 = 'ADC1 ENG Position angle [deg]'
  1208 = 'ADC1 OFF position angle [deg]'
  1559 = 'ADC1 OFF Position angle [deg]'
  186 = 'ADC1:'
  1634 = 'ADC2'
  338 = 'ADC2  ENG position angle [deg]'
  767 = 'ADC2  OFF position angle [deg]'
  192 = 'ADC2 OFF position angle [deg]'
  191 = 'ADC2:'
  795 = 'Additional information mostly used for description of errors'
  1700 = 'Alt :'
  1042 = 'Ambient'
  292 = 'Angles'
  2270 = 'Apparent Coordinates'
  2318 = 'Apparent Declination [ddmmss]'
  2453 = 'Apparent Declination [rad]'
  2121 = 'Apparent Right Ascension [hhmmss]'
  785 = 'Apparent Right Ascension [rad]'
  928 = 'Atmospheric Pressure [mbar]'
  933 = 'Atmospheric Relative Humidity [0..1]'
  943 = 'Atmospheric Temperature [deg C]'
  16 = 'AUTO'
  815 = 'Auto Disable'
  822 = 'Auto Disable Motor After Move'
  194 = 'Axes Status'
  127 = 'Axes2'
  938 = 'Axis Ready'
  22 = 'Axis Status'
  171 = 'Axis Type'
  1198 = 'Axis1'
  34 = 'Axis2'
  1709 = 'Az :'
  174 = 'Backlash'
  964 = 'BLUE = Used\nBLANK = Not Used'
  912 = 'Brake Active'
  507 = 'Brake Feedback Signal is Active Low'
  945 = 'Brake Used'
  173 = 'Brakes'
  177 = 'Brakes Used'
  824 = 'CCS Simulator'
  920 = 'CCS Simulator connected to ASTRO Module'
  794 = 'Check'
  869 = 'Check the box if this is an SoE drive (Sercos over EtherCAT) , e.g. AX5000'
  176 = 'Cicular-Optimised'
  175 = 'Circular-Opt'
  836 = 'Clear NOVRAM'
  843 = 'Clear NOVRAM. Use it with care!\n\nThis is needed ONLY if NOVRAM was previously used for data structures different than T_MOTOR_CFG (or for previous versions of T_MOTOR_CFG).\nBring the motor to NOT_READY first and then clear NOVRAM.'
  932 = 'Controller Enabled'
  180 = 'Coordinates'
  903 = 'Dec :'
  595 = 'Dec:'
  1067 = 'Declination [ddmmss]'
  1663 = 'Default Vel:'
  621 = 'Deg'
  1478 = 'Deg:'
  325 = 'Deterministic Data [rad]'
  763 = 'DISABLE'
  1003 = 'DISABLE\nAXIS'
  1770 = 'DROT'
  1640 = 'DROT :'
  405 = 'DROT control'
  1596 = 'DROT Control'
  1569 = 'DROT Moor'
  498 = 'DROT Motor'
  673 = 'DROT position angle [deg]'
  1631 = 'DROT position [deg]'
  399 = 'DROT Status'
  2033 = 'Dut:'
  403 = 'ELEV'
  619 = 'ELEV mode (3)'
  179 = 'Elevation Mode:  WHITE=Not Active\nGREEN=Activated'
  522 = 'ELEVK'
  866 = 'ENABLE'
  997 = 'ENABLE\nAXIS'
  867 = 'Enable Clear NOVRAM'
  847 = 'Enabled'
  187 = 'ENG'
  1781 = 'eng'
  909 = 'ENG (HOME) mode (=1)'
  364 = 'ENG mode (0)'
  1235 = 'ENG mode (=0)'
  597 = 'Engineering mode (0)'
  188 = 'Engineering mode (=0)'
  1019 = 'Engineering Mode \\nWHITE=Not active\nGREEN=Activated'
  2185 = 'Engineering Mode:  WHITE=Not active\nGREEN=Activated'
  1092 = 'Engineering ModeWHITE=Not active\nGREEN=Activated'
  1794 = 'Equinox'
  520 = 'Equinox:'
  851 = 'Error'
  870 = 'ERROR'
  12 = 'Error Description'
  861 = 'Error ID'
  806 = 'Event'
  1562 = 'Field Rotation :'
  2763 = 'Field Rotation [deg]'
  787 = 'Flag if motor is locked'
  951 = 'GREEN = Enabled\nRED = Disabled'
  990 = 'GREEN = In Position\nBLANK = Not In Position (or not used)'
  925 = 'GREEN = Initialised\nRED = Not Initialised'
  958 = 'GREEN = Ready\nRED = Not Ready'
  846 = 'GREEN=Enabled\nRED=NOT Enabled'
  848 = 'GREEN=Initialised\nRED=NOT Initialised'
  2465 = 'HA'
  678 = 'HA :'
  2560 = 'Hour Angle [deg]'
  96 = 'Hour Angle [rad]'
  918 = 'Humidity :'
  750 = 'Humidity [%]'
  801 = "If active, check if the in-pos signal is active after the move completes. If it is not, it's a failure."
  2525 = 'If active, it is not safe to operate the motor.'
  808 = 'If checked, In-Position feedback signal is active low'
  888 = 'If GREEN, tracking is OK'
  759 = 'If the motor is locked, during INIT the motor will not move and its position will be set to this value.'
  984 = 'In Position'
  829 = 'In-Pos Check'
  166 = 'INDEX'
  865 = 'INIT'
  162 = 'INIT Sequence Definition'
  516 = 'INIT sequence timeout in [ms].'
  971 = 'INIT Step'
  514 = 'INIT:'
  845 = 'Initialised'
  871 = 'INITIALIZING'
  924 = 'Lapse Rate'
  395 = 'Lapserate:'
  859 = 'Leap Second:'
  168 = 'LHW'
  812 = 'Local Control'
  181 = 'Local Sidereal Time'
  1751 = 'Local Sidereal Time [h]'
  854 = 'Local Time:'
  752 = 'Lock'
  965 = 'LST'
  894 = 'LST :'
  169 = 'LSTOP'
  1066 = 'Max Vel:'
  513 = 'Max:'
  531 = 'Mean Coordinates'
  998 = 'Mean Declination [ddmmss]'
  2704 = 'Mean Right Ascension [hhmmss]'
  512 = 'Min:'
  13 = 'Mode Control'
  855 = 'Mode:'
  591 = 'Motor 1 target position in user units (UU).'
  2145 = 'Motor 2 target position in user units (UU).'
  862 = 'Motor Status'
  1653 = 'Motor.library ver. %s'
  769 = 'MOVE ABS'
  610 = 'MOVE REL'
  775 = 'MOVE VEL+'
  605 = 'MOVE VEL-'
  515 = 'MOVE:'
  875 = 'MOVING'
  103 = 'Nord:'
  1494 = 'North Angle :'
  630 = 'North Angle [deg]'
  146 = 'North angle [deg]'
  104 = 'North angle [rad]'
  838 = 'NOT READY'
  646 = 'Observed Coordinates'
  1654 = 'Observed Declination [ddmmss]'
  1128 = 'Observed Right Ascension [hhmmss]'
  17 = 'OFF'
  2399 = 'OFF (HOME) mode (1)'
  184 = 'OFF (HOME) mode (=1)'
  1168 = 'Offset (REL)'
  893 = 'OK'
  1674 = 'PA :'
  2919 = 'Paralacti :'
  467 = 'Paralactic :'
  1847 = 'Parallactic :'
  1666 = 'Parallactic Angle [deg]'
  205 = 'Parallactic Angle [rad]'
  2083 = 'Pos:'
  20 = 'Posang:'
  1202 = 'PosAngle'
  1127 = 'Position'
  1376 = 'Position (ABS)'
  906 = 'Position angle [deg]'
  773 = 'Position:'
  509 = 'Positive, negative or zero (no backlash)'
  731 = 'POST-INIT'
  745 = 'POST-MOVE'
  724 = 'PRE-INIT'
  738 = 'PRE-MOVE'
  210 = 'Pressure'
  913 = 'Pressure :'
  2321 = 'Pressure [mbar]'
  1012 = 'Pressure:'
  887 = 'Pupil :'
  2295 = 'Pupil Angle :'
  230 = 'Pupil Angle [deg]'
  1253 = 'Pupil angle[deg]'
  56 = 'Pupil angle[rad]'
  955 = 'Pupil Rotation :'
  429 = 'Pupil Rotation [deg]'
  711 = 'Pupil:'
  1234 = 'Ra'
  898 = 'RA :'
  2102 = 'Ra :'
  596 = 'Ra:'
  1644 = 'Ready'
  872 = 'READY'
  919 = 'RED = Applied\nBLANK = Released'
  167 = 'REF'
  2351 = 'Relative offset used by "MOVE REL"'
  21 = 'RESET'
  2078 = 'Right Ascension[hhmmss]'
  977 = 'RPC Call Status'
  510 = 'Set'
  615 = 'SET POS'
  873 = 'SETTING \nPOSITION'
  511 = 'Setting both limits to 0 means that limits are not used.'
  400 = 'SKY'
  534 = 'SKY mode (2)'
  521 = 'Sky Mode:  WHITE=Not Active\nGREEN=Activated'
  1200 = 'SKYO'
  868 = 'SoE Drive'
  1111 = 'Speed (Pos)'
  1135 = 'Speed (Vel)'
  874 = 'STANDSTILL'
  401 = 'STAT'
  2172 = 'STAT mode (1)'
  782 = 'State'
  864 = 'State:'
  1877 = 'Stationary Mode:  WHITE=Not Active\nGREEN=Activated'
  850 = 'Status'
  800 = 'Status Description'
  863 = 'Status:'
  10 = 'STOP'
  530 = 'STOPPING'
  788 = 'Substate'
  1869 = 'Substate:'
  172 = 'SW Limits'
  517 = 'Switch exit timeout in [ms].'
  518 = 'SWITCH:'
  601 = 'Switches'
  163 = 'Switches \nActive Low'
  448 = 'TAI time [sec]'
  331 = 'TAI:'
  433 = 'Target'
  1119 = 'Target              Actual'
  2440 = 'Target Position [deg]'
  1683 = 'TEL Altitude [deg]'
  648 = 'TEL Altitude [rad]'
  1692 = 'TEL Azimuth [deg]'
  2490 = 'TEL Azimuth [rad]'
  948 = 'TEL Dec'
  939 = 'TEL RA'
  2128 = 'Temperaature'
  1440 = 'Temperaature:'
  908 = 'Temperature :'
  254 = 'Temperature [degC]'
  1727 = 'Temperature:'
  766 = 'The motor will not move, if the target position is closer to the locked position than this value.'
  741 = 'Time'
  1211 = 'Time mode [UTC, Local or Simulation]'
  858 = 'Time Mode:'
  170 = 'Timeouts [ms]'
  780 = 'Tolerance:'
  1172 = 'Total Offset :'
  2457 = 'Tracking Data'
  1193 = 'Tracking mode (2)'
  1216 = 'Tracking mode (=2)'
  1630 = 'Tracking mode (=3)'
  165 = 'UHW'
  2048 = 'Unsafe'
  1219 = 'Unsafe !!!'
  1948 = 'Unsafe!'
  404 = 'USER'
  717 = 'User \nProcs'
  733 = 'User Data [hh/ddmmss, deg]'
  1645 = 'User defined Mode: WHITE=Not Active\nGREEN=Activated'
  1917 = 'USER mode (4)'
  1009 = "User Units: '%s'"
  164 = 'USTOP'
  1264 = 'UTC time'
  907 = 'UTC time [sec]'
  853 = 'UTC:'
  344 = 'Value 1'
  345 = 'Value 2'
  189 = 'Vel:'
  190 = 'Velocity for Engineering Mode [deg/sec]'
  18 = 'Velocity:'
  1016 = 'Ver: %s'
  402 = 'VLTI'
  95 = 'Wavelenght'
  972 = 'Wavelenghth:'
  1720 = 'Wavelength:'
  856 = 'WHITE=Not active\nGREEN=Activated'
  857 = 'WHITE=Not Active\nGREEN=Activated'
  19 = '[deg/sec]'
  15 = '[deg]'
END_TEXTLIST

// ---- VISUs/Astro/GUI_ASTRO_CCS_SIM.TcVIS
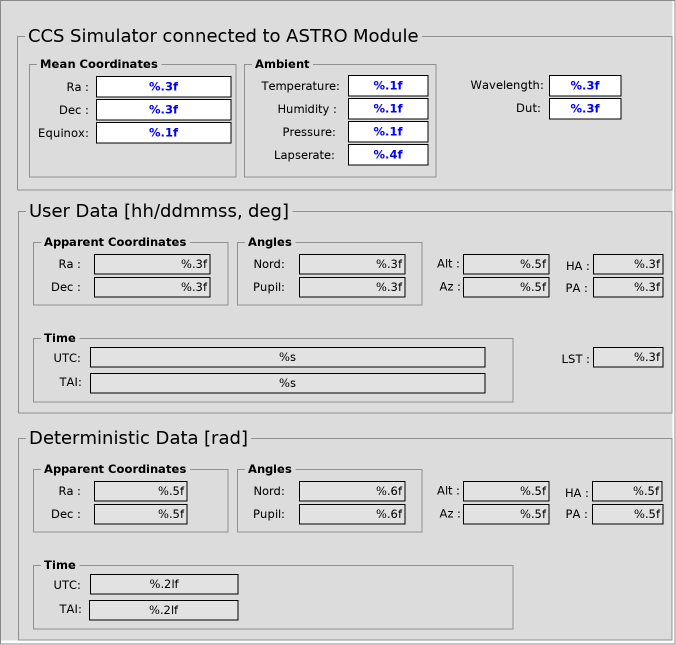
VISUALIZATION GUI_ASTRO_CCS_SIM  // 676x645
    Frame (0,0 676x645)
        shows GUI_TEMPLATE_ASTRO_CCS_SIM(m_DeviceName := 'astro', m_Instance := MAIN.astro)
END_VISUALIZATION

// ---- VISUs/Motor/GUI_Motor001_Cfg.TcVIS
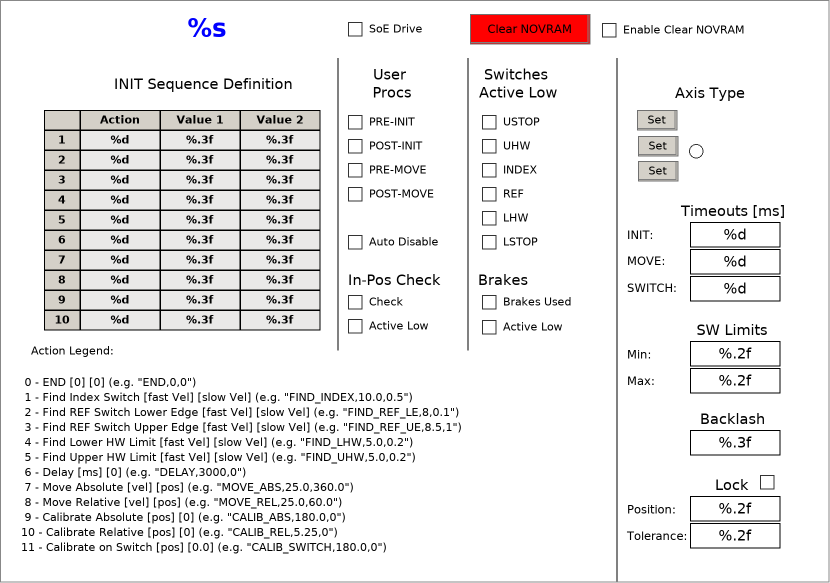
VISUALIZATION GUI_Motor001_Cfg  // 830x583
    Frame (0,0 828x581)
        shows GUI_TEMPLATE_MOTOR_CONFIG(m_Instance := MAIN.Motor001)
END_VISUALIZATION

// ---- VISUs/Motor/GUI_Motor002_Cfg.TcVIS
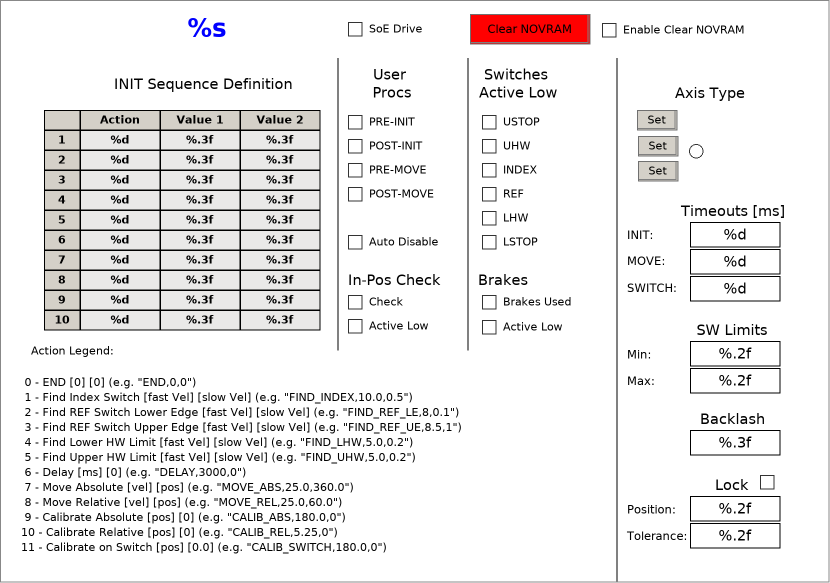
VISUALIZATION GUI_Motor002_Cfg  // 830x583
    Frame (0,0 828x581)
        shows GUI_TEMPLATE_MOTOR_CONFIG(m_Instance := MAIN.Motor002)
END_VISUALIZATION

// ---- VISUs/Motor/GUI_Motor001_Ctrl.TcVIS
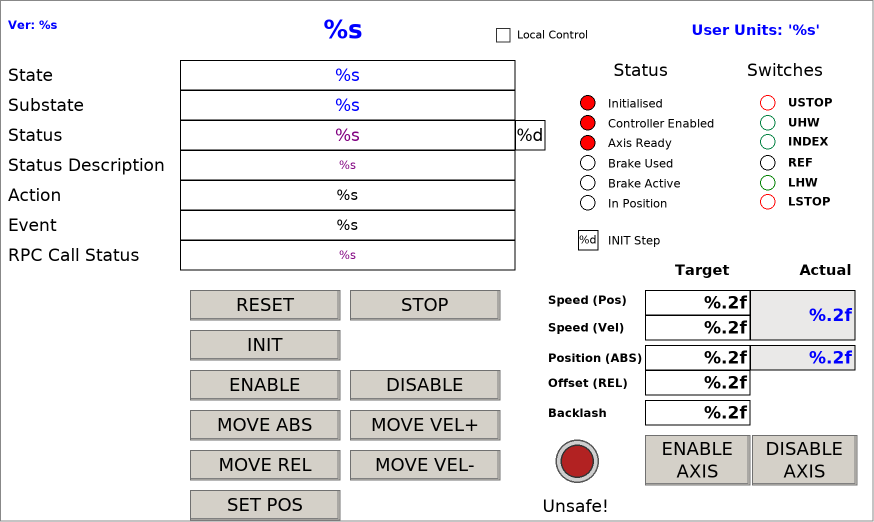
VISUALIZATION GUI_Motor001_Ctrl  // 874x522
    Frame (0,0 872x520)
        shows GUI_TEMPLATE_MOTOR_CONTROL(m_Instance := MAIN.Motor001)
END_VISUALIZATION

// ---- VISUs/Motor/GUI_Motor002_Ctrl.TcVIS
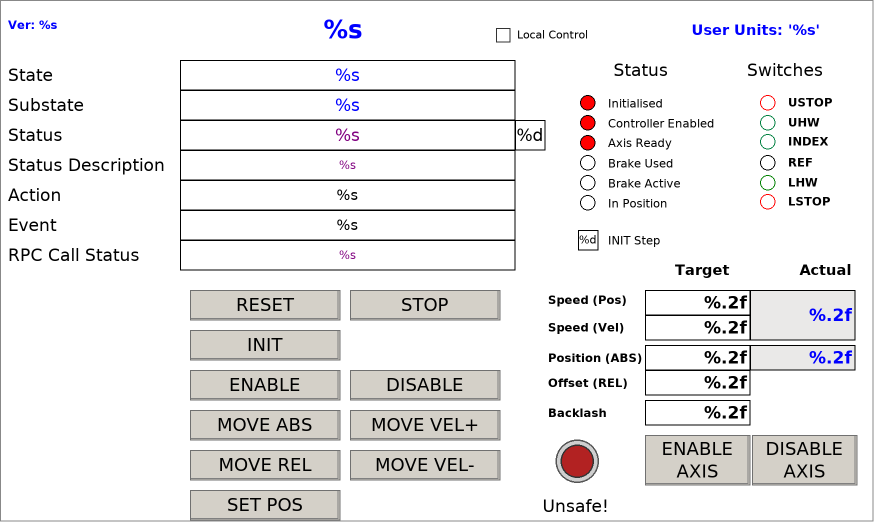
VISUALIZATION GUI_Motor002_Ctrl  // 874x522
    Frame (0,0 872x520)
        shows GUI_TEMPLATE_MOTOR_CONTROL(m_Instance := MAIN.Motor002)
END_VISUALIZATION

// ---- VISUs/Templates/GUI_TEMPLATE_ASTRO_CCS_SIM.TcVIS
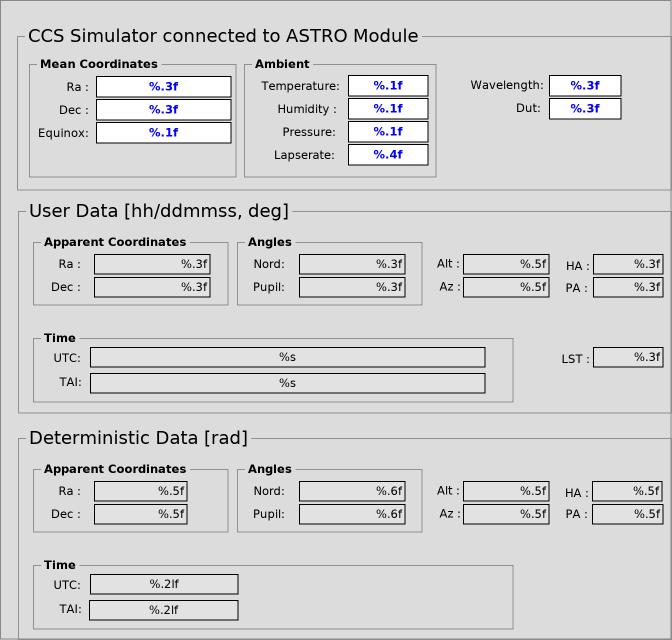
VISUALIZATION GUI_TEMPLATE_ASTRO_CCS_SIM  // 672x640
VAR_INPUT
	m_DeviceName : STRING;
END_VAR
VAR_IN_OUT
	m_Instance : FB_ASTRO;
END_VAR
    GroupBox (17,28 655x162), "CCS Simulator connected to ASTRO Module"
        GroupBox (12,28 207x121), "Mean Coordinates"
            Label (23,21 40x20), "Ra :"
            Label (23,44 40x20), "Dec :"
            Rectangle (67,20 135x21), "%.3f", tooltip "Mean Right Ascension [hhmmss]", text variable: m_Instance.AstroData.mean.alpha
                OnMouseDown: write the text variable via Edit
            Rectangle (67,43 135x21), "%.3f", tooltip "Mean Declination [ddmmss]", text variable: m_Instance.AstroData.mean.delta
                OnMouseDown: write the text variable via Edit
            Rectangle (67,66 135x21), "%.1f", tooltip "Equinox", text variable: m_Instance.AstroData.mean.equinox
                OnMouseDown: write the text variable via Edit
            Label (3,67 60x20), "Equinox:"
        GroupBox (227,28 192x121), "Ambient"
            Label (7,20 92x20), "Temperature:"
            Label (17,43 79x20), "Humidity :"
            Rectangle (104,19 80x21), "%.1f", tooltip "Temperature [degC]", text variable: m_Instance.AstroData.environment.temperature
                OnMouseDown: write the text variable via Edit
            Rectangle (104,42 80x21), "%.1f", tooltip "Humidity [%]", text variable: m_Instance.AstroData.environment.humidity
                OnMouseDown: write the text variable via Edit
            Rectangle (104,65 80x21), "%.1f", tooltip "Pressure [mbar]", text variable: m_Instance.AstroData.environment.pressure
                OnMouseDown: write the text variable via Edit
            Label (25,66 70x20), "Pressure:"
            Label (24,89 70x20), "Lapserate:"
            Rectangle (104,88 80x21), "%.4f", tooltip "Lapse Rate", text variable: m_Instance.AstroData.environment.lapserate
                OnMouseDown: write the text variable via Edit
        Rectangle (532,47 72x21), "%.3f", text variable: m_Instance.AstroData.wavelength
            OnMouseDown: write the text variable via Edit
        Rectangle (532,70 72x21), "%.3f", text variable: m_Instance.AstroData.dut
            OnMouseDown: write the text variable via Edit
        Label (481,70 46x20), "Dut:"
    GroupBox (18,203 654x210), "User Data [hh/ddmmss, deg]"
        GroupBox (15,31 195x71), "Apparent Coordinates"
            Label (11,20 40x20), "Ra :"
            Label (11,43 40x20), "Dec :"
            Label (8,70 60x20)
            Rectangle (61,43 116x20), "%.3f", tooltip "Apparent Declination [ddmmss]", text variable: m_Instance.AstroData.tracking_data.dec_dms
            Rectangle (61,20 116x20), "%.3f", tooltip "Apparent Right Ascension [hhmmss]", text variable: m_Instance.AstroData.tracking_data.ra_hms
        Rectangle (575,74 70x20), "%.3f", tooltip "Parallactic Angle [deg]", text variable: m_Instance.AstroData.tracking_data.pa_deg
        Label (523,75 50x20), "PA :"
        Label (408,51 37x19), "Alt :"
        Label (411,74 35x19), "Az :"
        GroupBox (219,31 185x71), "Angles"
            Label (11,20 40x20), "Nord:"
            Label (11,43 40x20), "Pupil:"
            Label (8,70 60x20)
            Rectangle (62,20 106x20), "%.3f", tooltip "North angle [deg]", text variable: m_Instance.UserPointingKernel.north_angle
            Rectangle (62,43 106x20), "%.3f", tooltip "Pupil angle[deg]", text variable: m_Instance.UserPointingKernel.pupil_angle
        Rectangle (445,74 86x20), "%.5f", tooltip "TEL Azimuth [deg]", text variable: m_Instance.AstroData.tracking_data.az_deg
        Rectangle (445,51 86x20), "%.5f", tooltip "TEL Altitude [deg]", text variable: m_Instance.AstroData.tracking_data.alt_deg
        GroupBox (15,127 480x72), "Time"
            Label (11,18 40x20), "UTC:"
            Label (6,42 46x20), "TAI:"
            Label (8,70 60x20)
            Rectangle (57,17 395x20), "%s", tooltip "UTC time", text variable: m_Instance.in_TimeStat.sUtcTime
            Rectangle (57,43 395x20), "%s", tooltip "TAI time [sec]", text variable: m_Instance.in_TimeStat.sTaiTime
        Label (534,146 41x20), "LST :"
        Label (533,280 41x20), "HA :"
    Label (464,75 83x20), "Wavelength:"
    Label (552,256 41x20), "HA :"
    Rectangle (593,254 70x20), "%.3f", tooltip "Hour Angle [deg]", text variable: m_Instance.AstroData.tracking_data.ha_deg
    GroupBox (18,430 654x210), "Deterministic Data [rad]"
        GroupBox (15,31 195x71), "Apparent Coordinates"
            Label (11,20 40x20), "Ra :"
            Label (11,43 40x20), "Dec :"
            Label (8,70 60x20)
            Rectangle (61,43 93x20), "%.5f", tooltip "Apparent Declination [rad]", text variable: m_Instance.AstroData.tracking_data.dec_r
            Rectangle (61,20 93x20), "%.5f", tooltip "Apparent Right Ascension [rad]", text variable: m_Instance.AstroData.tracking_data.ra_r
        Rectangle (574,74 71x20), "%.5f", tooltip "Parallactic Angle [rad]", text variable: m_Instance.AstroData.tracking_data.pa_r
        Label (523,74 50x20), "PA :"
        Label (408,51 37x19), "Alt :"
        Label (411,74 35x19), "Az :"
        GroupBox (219,31 185x71), "Angles"
            Label (11,20 40x20), "Nord:"
            Label (11,43 40x20), "Pupil:"
            Label (8,70 60x20)
            Rectangle (62,20 106x20), "%.6f", tooltip "North angle [rad]", text variable: m_Instance.q_trk_data.north_angle
            Rectangle (62,43 106x20), "%.6f", tooltip "Pupil angle[rad]", text variable: m_Instance.q_trk_data.pupil_angle
        Rectangle (445,74 86x20), "%.5f", tooltip "TEL Azimuth [rad]", text variable: m_Instance.AstroData.tracking_data.az_r
        Rectangle (445,51 86x20), "%.5f", tooltip "TEL Altitude [rad]", text variable: m_Instance.AstroData.tracking_data.alt_r
        GroupBox (15,127 480x72), "Time"
            Label (11,18 40x20), "UTC:"
            Label (6,42 46x20), "TAI:"
            Label (8,70 60x20)
            Rectangle (57,17 148x20), "%.2lf", tooltip "UTC time [sec]", text variable: m_Instance.out_CcsDeterministic.time_utc
            Rectangle (56,43 149x20), "%.2lf", tooltip "TAI time [sec]", text variable: m_Instance.out_CcsDeterministic.time_tai
    Rectangle (593,347 70x20), "%.3f", tooltip "Local Sidereal Time [h]", text variable: m_Instance.out_CcsDeterministic.time_lst
    Rectangle (592,481 70x20), "%.5f", tooltip "Hour Angle [rad]", text variable: m_Instance.AstroData.tracking_data.ha_r
END_VISUALIZATION

// ---- VISUs/Templates/GUI_TEMPLATE_MA_DROT.TcVIS
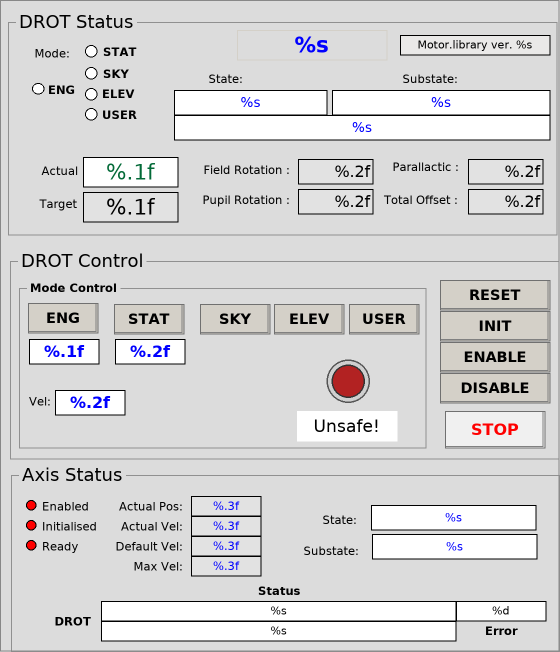
VISUALIZATION GUI_TEMPLATE_MA_DROT  // 560x652
VAR_INPUT
	m_DeviceName : STRING;
END_VAR
VAR_IN_OUT
	m_Instance : FB_MA_DROT;
END_VAR
    GroupBox (10,253 549x206), "DROT Control"
        Button (435,158 100x37), "STOP"
            OnMouseClick: execute { m_Instance.ctrl.nCommand:= E_MA_COMMAND.STOP; m_Instance.ctrl.bExecute:=(TRUE); }
        GroupBox (9,27 407x168), "Mode Control"
            Button (181,24 70x30), "SKY", tooltip "SKY mode (2)", input disabled if: NOT m_Instance.in_bSafe
                OnMouseClick: execute {
                    m_Instance.ctrl.nMode:= E_DROT_MODE.SKY;
                    m_Instance.ctrl.nCommand:=E_MA_COMMAND.START_TRACK;
                    m_Instance.ctrl.bExecute:=(TRUE);
                }
            Rectangle (10,59 70x25), "%.1f", tooltip "[deg]", text variable: m_Instance.ctrl.lrTargetPos
                OnMouseDown: write the text variable via Edit
            Button (9,23 70x30), "ENG", tooltip "Engineering mode (0)", input disabled if: NOT m_Instance.in_bSafe
                OnMouseClick: execute {
                    m_Instance.ctrl.nMode:= E_DROT_MODE.ENG;
                    m_Instance.ctrl.nCommand:= E_MA_COMMAND.STOP_TRACK;
                    m_Instance.ctrl.bExecute:=(TRUE);
                }
            Rectangle (36,110 70x25), "%.2f", tooltip "Velocity for Engineering Mode [deg/sec]", text variable: m_Instance.ctrl.lrTargetVel
                OnMouseDown: write the text variable via Edit
            Button (255,24 70x30), "ELEV", tooltip "ELEV mode (3)", input disabled if: NOT m_Instance.in_bSafe
                OnMouseClick: execute {
                    m_Instance.ctrl.nMode:= E_DROT_MODE.ELEV;
                    m_Instance.ctrl.nCommand:=E_MA_COMMAND.START_TRACK;
                    m_Instance.ctrl.bExecute:=(TRUE);
                }
            Button (95,24 70x30), "STAT", tooltip "STAT mode (1)", input disabled if: NOT m_Instance.in_bSafe
                OnMouseClick: execute {
                    m_Instance.ctrl.nMode:=E_DROT_MODE.STAT;
                    m_Instance.ctrl.nCommand:= E_MA_COMMAND.STOP_TRACK;
                    m_Instance.ctrl.bExecute:=(TRUE);
                }
            Button (330,24 70x30), "USER", tooltip "USER mode (4)", input disabled if: NOT m_Instance.in_bSafe
                OnMouseClick: execute {
                    m_Instance.ctrl.nMode:= E_DROT_MODE.USER;
                    m_Instance.ctrl.nCommand:=E_MA_COMMAND.START_TRACK;
                    m_Instance.ctrl.bExecute:=(TRUE);
                }
            Label (5,109 30x25), "Vel:"
            Rectangle (96,59 70x25), "%.2f", tooltip "Position angle [deg]", text variable: m_Instance.ctrl.lrPosang
                OnMouseDown: write the text variable via Edit
            Lamp1 (304,76 50x50), tooltip "If active, it is not safe to operate the motor.", variable: NOT m_Instance.in_bSafe, invisible if: m_Instance.in_bSafe, style: Lamp-Lamp1-Red
            Rectangle (278,131 100x30), "Unsafe!", invisible if: m_Instance.in_bSafe
        Button (430,120 110x30), "DISABLE", input disabled if: NOT m_Instance.in_bSafe
            OnMouseClick: execute { m_Instance.ctrl.nCommand:= E_MA_COMMAND.DISABLE; m_Instance.ctrl.bExecute:=(TRUE); }
        Button (430,27 110x30), "RESET", input disabled if: NOT m_Instance.in_bSafe
            OnMouseClick: execute { m_Instance.ctrl.nCommand:= E_MA_COMMAND.RESET; m_Instance.ctrl.bExecute:=(TRUE); }
        Button (430,89 110x30), "ENABLE", input disabled if: NOT m_Instance.in_bSafe
            OnMouseClick: execute { m_Instance.ctrl.nCommand:= E_MA_COMMAND.ENABLE; m_Instance.ctrl.bExecute:=(TRUE); }
        Button (430,58 110x30), "INIT", input disabled if: NOT m_Instance.in_bSafe
            OnMouseClick: execute { m_Instance.ctrl.nCommand:= E_MA_COMMAND.INIT; m_Instance.ctrl.bExecute:=(TRUE); }
    GroupBox (11,467 549x185), "Axis Status"
        Label (105,27 70x25), "Actual Pos:"
        Rectangle (180,29 70x20), "%.3f", tooltip "[deg]", text variable: m_Instance.pMotor1^.stat.lrPosActual
        Rectangle (180,49 70x20), "%.3f", tooltip "[deg/sec]", text variable: m_Instance.pMotor1^.stat.lrVelActual
        Label (28,52 70x15), "Initialised"
        Ellipse (15,33 10x10), tooltip "GREEN=Enabled RED=NOT Enabled", colour toggle: (m_Instance.pMotor1^.stat.bEnabled) <> 0
        Label (28,32 70x15), "Enabled"
        Ellipse (15,53 10x10), tooltip "GREEN=Initialised RED=NOT Initialised", colour toggle: (m_Instance.pMotor1^.stat.bInitialised) <> 0
        Label (105,47 70x25), "Actual Vel:"
        Label (216,114 105x20), "Status"
        Label (438,154 105x20), "Error"
        Rectangle (90,154 355x20), "%s", tooltip "Error Description", text variable: m_Instance.pMotor1^.stat.sErrorText
        Label (28,142 55x25), "DROT"
        Label (28,72 70x15), "Ready"
        Ellipse (15,73 10x10), tooltip "GREEN=Initialised RED=NOT Initialised", colour toggle: (m_Instance.pMotor1^.stat.bAxisReady) <> 0
        Rectangle (90,134 355x20), "%s", tooltip "Motor Status", text variable: m_Instance.pMotor1^.stat.sStatus
        Rectangle (445,134 90x20), "%d", tooltip "Error ID", text variable: m_Instance.pMotor1^.stat.nErrorCode
        Label (105,67 70x25), "Default Vel:"
        Rectangle (180,69 70x20), "%.3f", tooltip "[deg/sec]", text variable: m_Instance.pMotor1^.cfg.lrDefaultVelocity
        Rectangle (360,38 165x25), "%s", text variable: m_Instance.pMotor1^.stat.sState
        Label (259,38 90x30), "State:"
        Label (261,69 90x30), "Substate:"
        Rectangle (361,67 165x25), "%s", text variable: m_Instance.pMotor1^.stat.sSubstate
        Label (105,87 70x25), "Max Vel:"
        Rectangle (180,89 70x20), "%.3f", tooltip "[deg/sec]", text variable: m_Instance.pMotor1^.stat.axis.lrMaxVelocity
    GroupBox (8,14 549x221), "DROT Status"
        Label (10,26 69x27), "Mode:"
        Ellipse (24,69 12x11), tooltip "Engineering Mode: WHITE=Not active GREEN=Activated", colour toggle: (m_Instance.stat.nMode) = E_DROT_MODE.ENG
        Ellipse (77,31 12x12), tooltip "Stationary Mode: WHITE=Not Active GREEN=Activated", colour toggle: (m_Instance.stat.nMode) = E_DROT_MODE.STAT
        Label (37,67 83x18), "ENG"
        Ellipse (77,53 12x12), tooltip "Sky Mode: WHITE=Not Active GREEN=Activated", colour toggle: (m_Instance.stat.nMode) = E_DROT_MODE.SKY
        Ellipse (77,74 12x12), tooltip "Elevation Mode: WHITE=Not Active GREEN=Activated", colour toggle: (m_Instance.stat.nMode) = E_DROT_MODE.ELEV
        Label (91,70 43x20), "ELEV"
        Label (92,50 45x20), "SKY"
        Label (92,28 90x20), "STAT"
        Rectangle (460,145 75x25), "%.2f", tooltip "Parallactic Angle [deg]", text variable: m_Instance.ctrl.lrParallactic, invisible if: m_Instance.stat.nMode=E_DROT_MODE.STAT or m_Instance.stat.nMode=E_DROT_MODE.ENG
        Label (366,143 88x20), "Parallactic :", invisible if: m_Instance.stat.nMode=E_DROT_MODE.STAT or m_Instance.stat.nMode=E_DROT_MODE.ENG
        Rectangle (324,76 218x25), "%s", text variable: m_Instance.stat.sm.sSubstate
        Rectangle (166,76 153x25), "%s", text variable: m_Instance.stat.sm.sState
        Rectangle (166,101 376x25), "%s", text variable: m_Instance.stat.sStatus
        Label (193,50 45x30), "State:"
        Rectangle (392,21 150x20), "Motor.library ver. %s", text variable: m_Instance.stat.sLibVersion
        Rectangle (229,16 150x30), "%s", text variable: m_DeviceName
        Label (389,50 64x30), "Substate:"
        Rectangle (75,143 95x30), "%.1f", text variable: m_Instance.pMotor1^.stat.lrPosActual
        Label (25,176 47x28), "Target"
        Rectangle (75,178 95x30), "%.1f", tooltip "Target Position [deg]", text variable: m_Instance.stat.lrPos
        Label (26,143 47x28), "Actual"
        Ellipse (77,94 12x12), tooltip "User defined Mode: WHITE=Not Active GREEN=Activated", colour toggle: (m_Instance.stat.nMode) = E_DROT_MODE.USER
        Label (91,91 45x20), "USER"
        Rectangle (290,175 75x25), "%.2f", tooltip "Pupil Rotation [deg]", text variable: m_Instance.ctrl.lrPupil, invisible if: m_Instance.stat.nMode=E_DROT_MODE.STAT or m_Instance.stat.nMode=E_DROT_MODE.ENG
        Rectangle (290,145 75x25), "%.2f", tooltip "Field Rotation [deg]", text variable: m_Instance.ctrl.lrRotation, invisible if: m_Instance.stat.nMode=E_DROT_MODE.STAT or m_Instance.stat.nMode=E_DROT_MODE.ENG
        Label (194,146 91x20), "Field Rotation :", invisible if: m_Instance.stat.nMode=E_DROT_MODE.STAT or m_Instance.stat.nMode=E_DROT_MODE.ENG
        Label (189,176 96x20), "Pupil Rotation :", invisible if: m_Instance.stat.nMode=E_DROT_MODE.STAT or m_Instance.stat.nMode=E_DROT_MODE.ENG
        Label (365,176 88x20), "Total Offset :", invisible if: m_Instance.stat.nMode=E_DROT_MODE.STAT or m_Instance.stat.nMode=E_DROT_MODE.ENG
        Rectangle (460,175 75x25), "%.2f", tooltip "Parallactic Angle [deg]", text variable: m_Instance.stat.lrTotalOffset, invisible if: m_Instance.stat.nMode=E_DROT_MODE.STAT or m_Instance.stat.nMode=E_DROT_MODE.ENG
END_VISUALIZATION

// ---- VISUs/Templates/GUI_TEMPLATE_MA_ADC.TcVIS
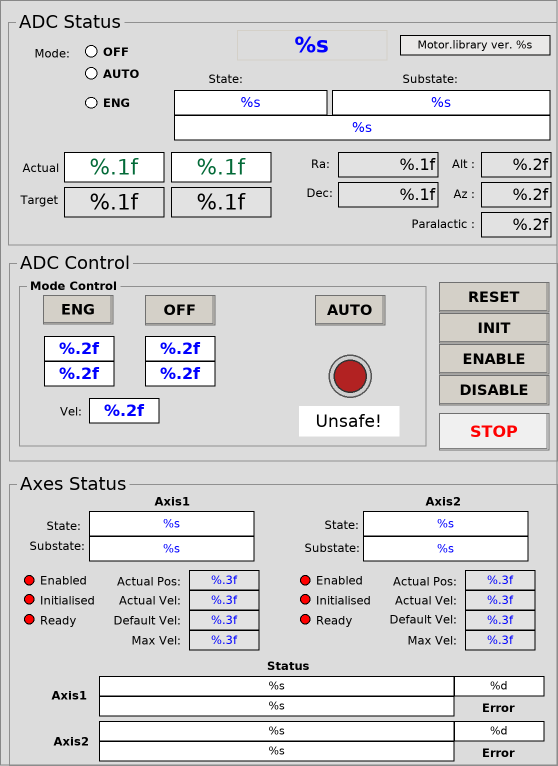
VISUALIZATION GUI_TEMPLATE_MA_ADC  // 558x766
VAR_INPUT
	m_DeviceName : STRING;
END_VAR
VAR_IN_OUT
	m_Instance : FB_MA_ADC;
END_VAR
    GroupBox (9,255 549x206), "ADC Control"
        Button (430,158 110x37), "STOP"
            OnMouseClick: execute { m_Instance.ctrl.nCommand:= E_MA_COMMAND.STOP; m_Instance.ctrl.bExecute:=(TRUE); }
        GroupBox (10,23 407x168), "Mode Control"
            Button (296,17 70x30), "AUTO", tooltip "Tracking mode (2)", input disabled if: NOT m_Instance.in_bSafe
                OnMouseClick: execute {
                    m_Instance.ctrl.nMode:= E_ADC_MODE.AUTO;
                    m_Instance.ctrl.nCommand:=E_MA_COMMAND.START_TRACK;
                    m_Instance.ctrl.bExecute:=(TRUE);
                }
            Rectangle (70,120 70x25), "%.2f", tooltip "Velocity for Engineering Mode [deg/sec]", text variable: m_Instance.ctrl.lrTargetVel
                OnMouseDown: write the text variable via Edit
            Button (126,17 70x30), "OFF", tooltip "OFF (HOME) mode (1)", input disabled if: NOT m_Instance.in_bSafe
                OnMouseClick: execute {
                    m_Instance.ctrl.nMode:=E_ADC_MODE.OFF;
                    m_Instance.ctrl.nCommand:= E_MA_COMMAND.STOP_TRACK;
                    m_Instance.ctrl.bExecute:=(TRUE);
                }
            Label (36,121 30x25), "Vel:"
            Rectangle (126,58 70x25), "%.2f", tooltip "ADC1 OFF Position angle [deg]", text variable: m_Instance.ctrl.lrPosang[1]
                OnMouseDown: write the text variable via Edit
            Rectangle (126,83 70x25), "%.2f", tooltip "ADC2 OFF position angle [deg]", text variable: m_Instance.ctrl.lrPosang[2]
                OnMouseDown: write the text variable via Edit
            Button (24,17 70x29), "ENG", tooltip "ENG mode (0)", input disabled if: NOT m_Instance.in_bSafe
                OnMouseClick: execute {
                    m_Instance.ctrl.nMode:=E_ADC_MODE.ENG;
                    m_Instance.ctrl.nCommand:= E_MA_COMMAND.STOP_TRACK;
                    m_Instance.ctrl.bExecute:=(TRUE);
                }
            Rectangle (25,58 70x25), "%.2f", tooltip "ADC1 ENG Position angle [deg]", text variable: m_Instance.ctrl.lrTargetPos[1]
                OnMouseDown: write the text variable via Edit
            Lamp1 (306,73 50x50), tooltip "If active, it is not safe to operate the motor.", variable: NOT m_Instance.in_bSafe, invisible if: m_Instance.in_bSafe, style: Lamp-Lamp1-Red
        Button (430,120 110x30), "DISABLE", input disabled if: NOT m_Instance.in_bSafe
            OnMouseClick: execute { m_Instance.ctrl.nCommand:= E_MA_COMMAND.DISABLE; m_Instance.ctrl.bExecute:=(TRUE); }
        Button (430,27 110x30), "RESET", input disabled if: NOT m_Instance.in_bSafe
            OnMouseClick: execute { m_Instance.ctrl.nCommand:= E_MA_COMMAND.RESET; m_Instance.ctrl.bExecute:=(TRUE); }
        Button (430,89 110x30), "ENABLE", input disabled if: NOT m_Instance.in_bSafe
            OnMouseClick: execute { m_Instance.ctrl.nCommand:= E_MA_COMMAND.ENABLE; m_Instance.ctrl.bExecute:=(TRUE); }
        Button (430,58 110x30), "INIT", input disabled if: NOT m_Instance.in_bSafe
            OnMouseClick: execute { m_Instance.ctrl.nCommand:= E_MA_COMMAND.INIT; m_Instance.ctrl.bExecute:=(TRUE); }
    GroupBox (9,476 549x290), "Axes Status"
        Label (98,93 77x25), "Actual Pos:"
        Rectangle (180,94 70x20), "%.3f", tooltip "[deg]", text variable: m_Instance.pMotor1^.stat.lrPosActual
        Rectangle (180,114 70x20), "%.3f", tooltip "[deg/sec]", text variable: m_Instance.pMotor1^.stat.lrVelActual
        Label (28,117 70x15), "Initialised"
        Label (28,97 70x15), "Enabled"
        Ellipse (15,118 10x10), tooltip "GREEN=Initialised RED=NOT Initialised", colour toggle: (m_Instance.pMotor1^.stat.bInitialised) <> 0
        Label (105,112 70x25), "Actual Vel:"
        Label (227,180 105x20), "Status"
        Label (437,222 105x20), "Error"
        Rectangle (90,220 355x20), "%s", tooltip "Error Description", text variable: m_Instance.pMotor1^.stat.sErrorText
        Label (28,137 70x15), "Ready"
        Ellipse (15,138 10x10), tooltip "GREEN=Initialised RED=NOT Initialised", colour toggle: (m_Instance.pMotor1^.stat.bAxisReady) <> 0
        Rectangle (90,200 355x20), "%s", tooltip "Motor Status", text variable: m_Instance.pMotor1^.stat.sStatus
        Rectangle (445,200 90x20), "%d", tooltip "Error ID", text variable: m_Instance.pMotor1^.stat.nErrorCode
        Label (94,132 81x25), "Default Vel:"
        Rectangle (180,134 70x20), "%.3f", tooltip "[deg/sec]", text variable: m_Instance.pMotor1^.cfg.lrDefaultVelocity
        Rectangle (80,35 165x25), "%s", text variable: m_Instance.pMotor1^.stat.sState
        Label (12,55 67x30), "Substate:"
        Rectangle (90,245 355x20), "%s", tooltip "Motor Status", text variable: m_Instance.pMotor2^.stat.sStatus
        Label (29,35 46x30), "State:"
        Label (437,267 105x20), "Error"
        Rectangle (354,35 165x25), "%s", text variable: m_Instance.pMotor2^.stat.sState
        Rectangle (80,60 165x25), "%s", text variable: m_Instance.pMotor1^.stat.sSubstate
        Rectangle (354,60 165x25), "%s", text variable: m_Instance.pMotor2^.stat.sSubstate
        Label (287,57 67x30), "Substate:"
        Label (308,34 45x30), "State:"
        Label (136,13 55x25), "Axis1"
        Label (408,13 53x25), "Axis2"
        Label (26,207 55x25), "Axis1"
        Ellipse (15,99 10x10), tooltip "GREEN=Enabled RED=NOT Enabled", colour toggle: (m_Instance.pMotor1^.stat.bEnabled) <> 0
        Ellipse (291,118 10x10), tooltip "GREEN=Initialised RED=NOT Initialised", colour toggle: (m_Instance.pMotor2^.stat.bInitialised) <> 0
        Label (105,152 70x25), "Max Vel:"
        Label (381,152 70x25), "Max Vel:"
    GroupBox (8,14 549x231), "ADC Status"
        Label (10,26 69x27), "Mode:"
        Ellipse (77,83 12x11), tooltip "Engineering Mode: WHITE=Not active GREEN=Activated", colour toggle: (m_Instance.stat.nMode) = E_ADC_MODE.ENG
        Ellipse (77,31 12x12), tooltip "Stationary Mode: WHITE=Not Active GREEN=Activated", colour toggle: (m_Instance.stat.nMode) = E_ADC_MODE.OFF
        Label (92,80 35x18), "ENG"
        Ellipse (77,53 12x12), tooltip "Sky Mode: WHITE=Not Active GREEN=Activated", colour toggle: (m_Instance.stat.nMode) = E_ADC_MODE.AUTO
        Label (92,28 90x20), "OFF"
        Label (285,140 40x20), "Ra:", invisible if: m_Instance.stat.nMode<>E_ADC_MODE.AUTO
        Label (288,169 40x20), "Dec:", invisible if: m_Instance.stat.nMode<>E_ADC_MODE.AUTO
        Rectangle (330,138 100x25), "%.1f", tooltip "TEL RA", text variable: m_Instance.stat.lrRa, invisible if: m_Instance.stat.nMode<>E_ADC_MODE.AUTO
        Rectangle (330,168 100x25), "%.1f", tooltip "TEL Dec", text variable: m_Instance.stat.lrDec, invisible if: m_Instance.stat.nMode<>E_ADC_MODE.AUTO
        Rectangle (473,198 70x25), "%.2f", tooltip "Parallactic Angle [deg]", text variable: m_Instance.stat.lrPa, invisible if: m_Instance.stat.nMode<>E_ADC_MODE.AUTO
        Label (372,200 98x20), "Paralactic :", invisible if: m_Instance.stat.nMode<>E_ADC_MODE.AUTO
        Rectangle (473,138 70x25), "%.2f", tooltip "TEL Altitude [deg]", text variable: m_Instance.stat.lrAlt, invisible if: m_Instance.stat.nMode<>E_ADC_MODE.AUTO
        Rectangle (473,168 70x25), "%.2f", tooltip "TEL Azimuth [deg]", text variable: m_Instance.stat.lrAz, invisible if: m_Instance.stat.nMode<>E_ADC_MODE.AUTO
        Label (420,140 50x20), "Alt :", invisible if: m_Instance.stat.nMode<>E_ADC_MODE.AUTO
        Label (420,170 50x20), "Az :", invisible if: m_Instance.stat.nMode<>E_ADC_MODE.AUTO
        Rectangle (324,76 218x25), "%s", text variable: m_Instance.stat.sm.sSubstate
        Rectangle (166,76 153x25), "%s", text variable: m_Instance.stat.sm.sState
        Rectangle (166,101 376x25), "%s", text variable: m_Instance.stat.sStatus
        Label (193,50 45x30), "State:"
        Rectangle (392,21 150x20), "Motor.library ver. %s", text variable: m_Instance.stat.sLibVersion
        Rectangle (229,16 150x30), "%s", text variable: m_DeviceName
        Label (389,50 64x30), "Substate:"
        Rectangle (56,138 100x30), "%.1f", text variable: m_Instance.pMotor1^.stat.lrPosActual
        Label (6,172 47x28), "Target"
        Rectangle (56,173 100x30), "%.1f", tooltip "Motor 1 target position in user units (UU).", text variable: m_Instance.pMotor1^.stat.lrPosTarget
        Label (7,140 47x28), "Actual"
        Label (92,50 45x20), "AUTO"
        Rectangle (163,138 100x30), "%.1f", text variable: m_Instance.pMotor2^.stat.lrPosActual
        Rectangle (163,173 100x30), "%.1f", tooltip "Motor 2 target position in user units (UU).", text variable: m_Instance.pMotor2^.stat.lrPosTarget
    Label (447,721 105x20), "Error"
    Rectangle (99,741 355x20), "%s", tooltip "Error Description", text variable: m_Instance.pMotor2^.stat.sErrorText
    Label (37,729 55x25), "Axis2"
    Rectangle (454,721 90x20), "%d", tooltip "Error ID", text variable: m_Instance.pMotor2^.stat.nErrorCode
    Label (382,569 78x25), "Actual Pos:"
    Rectangle (465,570 70x20), "%.3f", tooltip "[deg]", text variable: m_Instance.pMotor2^.stat.lrPosActual
    Rectangle (465,590 70x20), "%.3f", tooltip "[deg/sec]", text variable: m_Instance.pMotor2^.stat.lrVelActual
    Label (313,593 70x15), "Initialised"
    Label (313,573 70x15), "Enabled"
    Label (390,588 70x25), "Actual Vel:"
    Label (313,613 70x15), "Ready"
    Label (377,607 83x25), "Default Vel:"
    Rectangle (465,610 70x20), "%.3f", tooltip "[deg/sec]", text variable: m_Instance.pMotor2^.cfg.lrDefaultVelocity
    Ellipse (300,614 10x10), tooltip "GREEN=Initialised RED=NOT Initialised", colour toggle: (m_Instance.pMotor2^.stat.bAxisReady) <> 0
    Ellipse (300,575 10x10), tooltip "GREEN=Enabled RED=NOT Enabled", colour toggle: (m_Instance.pMotor2^.stat.bEnabled) <> 0
    Rectangle (44,361 70x25), "%.2f", tooltip "ADC2 ENG position angle [deg]", text variable: m_Instance.ctrl.lrTargetPos[2]
        OnMouseDown: write the text variable via Edit
    Rectangle (189,630 70x20), "%.3f", tooltip "[deg/sec]", text variable: m_Instance.pMotor1^.stat.axis.lrMaxVelocity
    Rectangle (465,630 70x20), "%.3f", tooltip "[deg/sec]", text variable: m_Instance.pMotor2^.stat.axis.lrMaxVelocity
    Rectangle (299,406 100x30), "Unsafe!", invisible if: m_Instance.in_bSafe
END_VISUALIZATION

// ---- VISUs/Templates/GUI_TEMPLATE_MOTOR_CONFIG.TcVIS
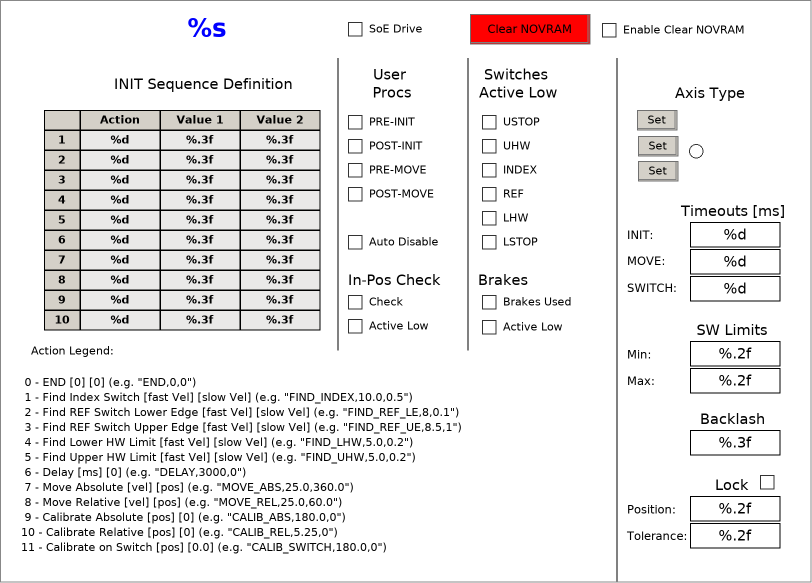
VISUALIZATION GUI_TEMPLATE_MOTOR_CONFIG  // 812x583
VAR_IN_OUT
	m_Instance : FB_MOTOR;
END_VAR
VAR
	bEnableNovramClear:	BOOL := FALSE;
END_VAR
    Label (28,336 150x30), "Action Legend:"
    Label (18,371 600x23), "0 - END [0] [0] (e.g. "END,0,0")"
    Label (18,386 600x23), "1 - Find Index Switch [fast Vel] [slow Vel] (e.g. "FIND_INDEX,10.0,0.5")"
    Label (18,401 600x23), "2 - Find REF Switch Lower Edge [fast Vel] [slow Vel] (e.g. "FIND_REF_LE,8,0.1")"
    Label (18,416 600x23), "3 - Find REF Switch Upper Edge [fast Vel] [slow Vel] (e.g. "FIND_REF_UE,8.5,1")"
    Label (18,431 600x23), "4 - Find Lower HW Limit [fast Vel] [slow Vel] (e.g. "FIND_LHW,5.0,0.2")"
    Label (18,446 600x23), "5 - Find Upper HW Limit [fast Vel] [slow Vel] (e.g. "FIND_UHW,5.0,0.2")"
    Label (18,476 600x23), "7 - Move Absolute [vel] [pos] (e.g. "MOVE_ABS,25.0,360.0")"
    Label (18,491 600x23), "8 - Move Relative [vel] [pos] (e.g. "MOVE_REL,25.0,60.0")"
    Label (18,506 600x23), "9 - Calibrate Absolute [pos] [0] (e.g. "CALIB_ABS,180.0,0")"
    Label (18,521 600x23), "10 - Calibrate Relative [pos] [0] (e.g. "CALIB_REL,5.25,0")"
    Label (18,461 600x23), "6 - Delay [ms] [0] (e.g. "DELAY,3000,0")"
    Label (18,536 600x23), "11 - Calibrate on Switch [pos] [0.0] (e.g. "CALIB_SWITCH,180.0,0")"
    Label (59,69 289x30), "INIT Sequence Definition"
    Label (462,54 113x59), "Switches Active Low"
    Checkbox (480,110 93x24), "USTOP", variable: m_Instance.cfg.bArrActiveLow[5].bValue, invisible if: false, input disabled if: false
    Checkbox (480,134 93x24), "UHW", variable: m_Instance.cfg.bArrActiveLow[4].bValue, invisible if: false, input disabled if: false
    Checkbox (480,158 93x24), "INDEX", variable: m_Instance.cfg.bArrActiveLow[3].bValue, invisible if: false, input disabled if: false
    Checkbox (480,182 93x24), "REF", variable: m_Instance.cfg.bArrActiveLow[2].bValue, invisible if: false, input disabled if: false
    Checkbox (480,206 93x24), "LHW", variable: m_Instance.cfg.bArrActiveLow[1].bValue, invisible if: false, input disabled if: false
    Checkbox (480,230 93x24), "LSTOP", variable: m_Instance.cfg.bArrActiveLow[0].bValue, invisible if: false, input disabled if: false
    Rectangle (87,7 240x42), "%s", text variable: m_Instance.sName
    Label (678,196 132x30), "Timeouts [ms]"
    Label (665,78 90x30), "Axis Type"
    Label (687,315 90x30), "SW Limits"
    Label (475,265 103x30), "Brakes"
    Label (685,404 95x30), "Backlash"
    RadioButton (687,112 114x78), variable: m_Instance.cfg.nAxisType-1, input disabled if: FALSE
        Areas[0]: Text=Linear
        Areas[1]: Text=Circular
        Areas[2]: Text=Circular-Opt
        p3166011961: Cicular-Optimised
    Checkbox (480,290 110x24), "Brakes Used", variable: m_Instance.cfg.bUseBrake, invisible if: false, input disabled if: false
    Checkbox (480,315 105x24), "Active Low", tooltip "Brake Feedback Signal is Active Low", variable: m_Instance.cfg.bActiveLowBrake, invisible if: false, input disabled if: false
    Rectangle (690,430 90x25), "%.3f", tooltip "Positive, negative or zero (no backlash)", text variable: m_Instance.cfg.lrBacklash
        OnMouseDown: write the text variable via Default
    Button (637,110 40x20), "Set"
        OnMouseClick: execute { m_Instance.cfg.nAxisType := 1; }
    Button (638,136 40x20), "Set"
        OnMouseClick: execute { m_Instance.cfg.nAxisType := 2; }
    Button (638,161 40x20), "Set"
        OnMouseClick: execute { m_Instance.cfg.nAxisType := 3; }
    Rectangle (690,341 90x25), "%.2f", tooltip "Setting both limits to 0 means that limits are not used.", text variable: m_Instance.cfg.lrMinPosition
        OnMouseDown: write the text variable via Default
    Rectangle (690,368 90x25), "%.2f", tooltip "Setting both limits to 0 means that limits are not used.", text variable: m_Instance.cfg.lrMaxPosition
        OnMouseDown: write the text variable via Default
    Label (624,340 37x29), "Min:"
    Label (624,366 37x30), "Max:"
    Label (624,220 49x30), "INIT:"
    Label (624,246 49x30), "MOVE:"
    Rectangle (690,222 90x25), "%d", tooltip "INIT sequence timeout in [ms].", text variable: m_Instance.cfg.nTimeoutInit
        OnMouseDown: write the text variable via Default
    Rectangle (690,249 90x25), "%d", tooltip "INIT sequence timeout in [ms].", text variable: m_Instance.cfg.nTimeoutMove
        OnMouseDown: write the text variable via Default
    Line (468,350) (468,58)
    Line (617,581) (617,58)
    Rectangle (690,276 90x25), "%d", tooltip "Switch exit timeout in [ms].", text variable: m_Instance.cfg.nTimeoutSwitch
        OnMouseDown: write the text variable via Default
    Label (624,273 60x30), "SWITCH:"
    Rectangle (80,110 80x20), "Action"
    Rectangle (160,110 80x20), "Value 1"
    Rectangle (240,110 80x20), "Value 2"
    Rectangle (44,130 36x20), "1"
    Rectangle (44,110 36x20)
    Rectangle (80,130 80x20), "%d", text variable: m_Instance.cfg.strArrInitSeq[1].nAction
        OnMouseDown: write the text variable via Default
    Rectangle (160,130 80x20), "%.3f", text variable: m_Instance.cfg.strArrInitSeq[1].lrValue1
        OnMouseDown: write the text variable via Default
    Rectangle (240,130 80x20), "%.3f", text variable: m_Instance.cfg.strArrInitSeq[1].lrValue2
        OnMouseDown: write the text variable via Default
    Rectangle (44,150 36x20), "2"
    Rectangle (80,150 80x20), "%d", text variable: m_Instance.cfg.strArrInitSeq[2].nAction
        OnMouseDown: write the text variable via Default
    Rectangle (160,150 80x20), "%.3f", text variable: m_Instance.cfg.strArrInitSeq[2].lrValue1
        OnMouseDown: write the text variable via Default
    Rectangle (240,150 80x20), "%.3f", text variable: m_Instance.cfg.strArrInitSeq[2].lrValue2
        OnMouseDown: write the text variable via Default
    Rectangle (44,170 36x20), "3"
    Rectangle (80,170 80x20), "%d", text variable: m_Instance.cfg.strArrInitSeq[3].nAction
        OnMouseDown: write the text variable via Default
    Rectangle (160,170 80x20), "%.3f", text variable: m_Instance.cfg.strArrInitSeq[3].lrValue1
        OnMouseDown: write the text variable via Default
    Rectangle (240,170 80x20), "%.3f", text variable: m_Instance.cfg.strArrInitSeq[3].lrValue2
        OnMouseDown: write the text variable via Default
    Rectangle (44,190 36x20), "4"
    Rectangle (80,190 80x20), "%d", text variable: m_Instance.cfg.strArrInitSeq[4].nAction
        OnMouseDown: write the text variable via Default
    Rectangle (160,190 80x20), "%.3f", text variable: m_Instance.cfg.strArrInitSeq[4].lrValue1
        OnMouseDown: write the text variable via Default
    Rectangle (240,190 80x20), "%.3f", text variable: m_Instance.cfg.strArrInitSeq[4].lrValue2
        OnMouseDown: write the text variable via Default
    Rectangle (44,210 36x20), "5"
    Rectangle (80,210 80x20), "%d", text variable: m_Instance.cfg.strArrInitSeq[5].nAction
        OnMouseDown: write the text variable via Default
    Rectangle (160,210 80x20), "%.3f", text variable: m_Instance.cfg.strArrInitSeq[5].lrValue1
        OnMouseDown: write the text variable via Default
    Rectangle (240,210 80x20), "%.3f", text variable: m_Instance.cfg.strArrInitSeq[5].lrValue2
        OnMouseDown: write the text variable via Default
    Rectangle (44,230 36x20), "6"
    Rectangle (80,230 80x20), "%d", text variable: m_Instance.cfg.strArrInitSeq[6].nAction
        OnMouseDown: write the text variable via Default
    Rectangle (160,230 80x20), "%.3f", text variable: m_Instance.cfg.strArrInitSeq[6].lrValue1
        OnMouseDown: write the text variable via Default
    Rectangle (240,230 80x20), "%.3f", text variable: m_Instance.cfg.strArrInitSeq[6].lrValue2
        OnMouseDown: write the text variable via Default
    Rectangle (44,250 36x20), "7"
    Rectangle (80,250 80x20), "%d", text variable: m_Instance.cfg.strArrInitSeq[7].nAction
        OnMouseDown: write the text variable via Default
    Rectangle (160,250 80x20), "%.3f", text variable: m_Instance.cfg.strArrInitSeq[7].lrValue1
        OnMouseDown: write the text variable via Default
    Rectangle (240,250 80x20), "%.3f", text variable: m_Instance.cfg.strArrInitSeq[7].lrValue2
        OnMouseDown: write the text variable via Default
    Rectangle (44,270 36x20), "8"
    Rectangle (80,270 80x20), "%d", text variable: m_Instance.cfg.strArrInitSeq[8].nAction
        OnMouseDown: write the text variable via Default
    Rectangle (160,270 80x20), "%.3f", text variable: m_Instance.cfg.strArrInitSeq[8].lrValue1
        OnMouseDown: write the text variable via Default
    Rectangle (240,270 80x20), "%.3f", text variable: m_Instance.cfg.strArrInitSeq[8].lrValue2
        OnMouseDown: write the text variable via Default
    Rectangle (44,290 36x20), "9"
    Rectangle (80,290 80x20), "%d", text variable: m_Instance.cfg.strArrInitSeq[9].nAction
        OnMouseDown: write the text variable via Default
    Rectangle (160,290 80x20), "%.3f", text variable: m_Instance.cfg.strArrInitSeq[9].lrValue1
        OnMouseDown: write the text variable via Default
    Rectangle (240,290 80x20), "%.3f", text variable: m_Instance.cfg.strArrInitSeq[9].lrValue2
        OnMouseDown: write the text variable via Default
    Rectangle (44,310 36x20), "10"
    Rectangle (80,310 80x20), "%d", text variable: m_Instance.cfg.strArrInitSeq[10].nAction
        OnMouseDown: write the text variable via Default
    Rectangle (160,310 80x20), "%.3f", text variable: m_Instance.cfg.strArrInitSeq[10].lrValue1
        OnMouseDown: write the text variable via Default
    Rectangle (240,310 80x20), "%.3f", text variable: m_Instance.cfg.strArrInitSeq[10].lrValue2
        OnMouseDown: write the text variable via Default
    Line (338,350) (338,58)
    Label (345,54 94x59), "User Procs"
    Checkbox (346,110 106x24), "PRE-INIT", variable: m_Instance.cfg.bExecUserPreInit, invisible if: false, input disabled if: false
    Checkbox (346,134 106x24), "POST-INIT", variable: m_Instance.cfg.bExecUserPostInit, invisible if: false, input disabled if: false
    Checkbox (346,158 106x24), "PRE-MOVE", variable: m_Instance.cfg.bExecUserPreMove, invisible if: false, input disabled if: false
    Checkbox (346,182 106x24), "POST-MOVE", variable: m_Instance.cfg.bExecUserPostMove, invisible if: false, input disabled if: false
    Label (687,470 90x30), "Lock"
    Rectangle (690,496 90x25), "%.2f", tooltip "If the motor is locked, during INIT the motor will not move and its position will be set to this value.", text variable: m_Instance.cfg.lrLockPos
        OnMouseDown: write the text variable via Default
    Rectangle (690,523 90x25), "%.2f", tooltip "The motor will not move, if the target position is closer to the locked position than this value.", text variable: m_Instance.cfg.lrLockTol
        OnMouseDown: write the text variable via Default
    Label (624,495 56x29), "Position:"
    Label (624,521 63x30), "Tolerance:"
    Checkbox (758,470 30x24), tooltip "Flag if motor is locked", variable: m_Instance.cfg.bLock, invisible if: false, input disabled if: false
    Checkbox (346,290 106x24), "Check", tooltip "If active, check if the in-pos signal is active after the move completes. If it is not, it's a failure.", variable: m_Instance.cfg.bCheckInPos, invisible if: false, input disabled if: false
    Checkbox (346,314 107x24), "Active Low", tooltip "If checked, In-Position feedback signal is active low", variable: m_Instance.cfg.bActiveLowInPos, invisible if: false, input disabled if: false
    Checkbox (346,230 127x24), "Auto Disable", tooltip "Auto Disable Motor After Move", variable: m_Instance.cfg.bDisableAfterMove, invisible if: false, input disabled if: false
    Label (345,265 103x30), "In-Pos Check"
    Button (470,14 120x30), "Clear NOVRAM", tooltip "Clear NOVRAM. Use it with care! This is needed ONLY if NOVRAM was previously used for data structures different than T_MOTOR_CFG (or for previous versions of T_MOTOR_CFG). Bring the motor to NOT_READY first and then clear NOVRAM.", input disabled if: bEnableNovramClear=false OR m_Instance.nNOVRAM_DevId=0
        OnMouseUp: execute {
            m_Instance.ctrl.bLocalCmd := TRUE;
            m_Instance.ctrl.nCommand:=E_MOTOR_COMMAND.CLEAR_NOVRAM;
            m_Instance.ctrl.bExecute:=(TRUE);
        }
    Checkbox (600,18 160x24), "Enable Clear NOVRAM", variable: bEnableNovramClear, invisible if: false, input disabled if: false
    Checkbox (346,17 90x24), "SoE Drive", tooltip "Check the box if this is an SoE drive (Sercos over EtherCAT) , e.g. AX5000", variable: m_Instance.cfg.bSoE_Drive, invisible if: false, input disabled if: false
END_VISUALIZATION

// ---- VISUs/Templates/GUI_TEMPLATE_MOTOR_CONTROL.TcVIS
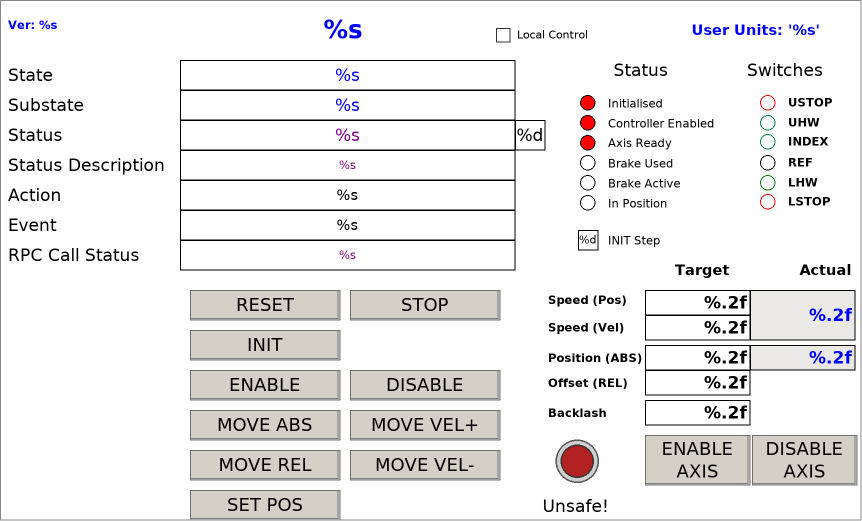
VISUALIZATION GUI_TEMPLATE_MOTOR_CONTROL  // 862x521
VAR_IN_OUT
	m_Instance:	FB_MOTOR;
END_VAR
    Rectangle (180,60 335x30), "%s", text variable: m_Instance.stat.sState
    Rectangle (180,90 335x30), "%s", text variable: m_Instance.stat.sSubstate
    Button (190,290 150x30), "RESET", input disabled if: NOT m_Instance.stat.bLocal OR NOT m_Instance.in_bSafe
        OnMouseDown: execute {
            m_Instance.ctrl.bLocalCmd := TRUE;
            m_Instance.ctrl.nCommand := E_MOTOR_COMMAND.RESET;
            m_Instance.ctrl.bExecute := TRUE;
        }
    Button (190,330 150x30), "INIT", input disabled if: NOT m_Instance.stat.bLocal OR NOT m_Instance.in_bSafe
        OnMouseDown: execute {
            m_Instance.ctrl.bLocalCmd := TRUE;
            m_Instance.ctrl.nCommand := E_MOTOR_COMMAND.INIT;
            m_Instance.ctrl.bExecute := TRUE;
        }
    Button (350,290 150x30), "STOP", input disabled if: NOT m_Instance.stat.bLocal OR NOT m_Instance.in_bSafe
        OnMouseDown: execute {
            m_Instance.ctrl.bLocalCmd := TRUE;
            m_Instance.ctrl.nCommand := E_MOTOR_COMMAND.STOP;
            m_Instance.ctrl.bExecute := TRUE;
        }
    Button (190,370 150x30), "ENABLE", input disabled if: NOT m_Instance.stat.bLocal OR NOT m_Instance.in_bSafe
        OnMouseDown: execute {
            m_Instance.ctrl.bLocalCmd := TRUE;
            m_Instance.ctrl.nCommand := E_MOTOR_COMMAND.ENABLE;
            m_Instance.ctrl.bExecute := TRUE;
        }
    Button (350,370 150x30), "DISABLE", input disabled if: NOT m_Instance.stat.bLocal OR NOT m_Instance.in_bSafe
        OnMouseDown: execute {
            m_Instance.ctrl.bLocalCmd := TRUE;
            m_Instance.ctrl.nCommand := E_MOTOR_COMMAND.DISABLE;
            m_Instance.ctrl.bExecute := TRUE;
        }
    Button (190,410 150x30), "MOVE ABS", input disabled if: NOT m_Instance.stat.bLocal OR NOT m_Instance.in_bSafe
        OnMouseDown: execute {
            m_Instance.ctrl.bLocalCmd := TRUE;
            m_Instance.ctrl.lrVelocity:=(m_Instance.cfg.lrDefaultVelocity);
            m_Instance.ctrl.nCommand := E_MOTOR_COMMAND.MOTOR_MOVE;
            m_Instance.ctrl.nMoveType := E_MOTOR_MOVE_TYPE.ABSOLUTE;
            m_Instance.ctrl.bExecute := TRUE;
        }
    Button (350,410 150x30), "MOVE VEL+", input disabled if: NOT m_Instance.stat.bLocal OR NOT m_Instance.in_bSafe
        OnMouseDown: execute {
            m_Instance.ctrl.bLocalCmd := TRUE;
            m_Instance.ctrl.nCommand := E_MOTOR_COMMAND.MOTOR_MOVE;
            m_Instance.ctrl.nMoveType := E_MOTOR_MOVE_TYPE.VELOCITY;
            m_Instance.ctrl.nDirection := MC_Positive_Direction;
            m_Instance.ctrl.bExecute := TRUE;
        }
    Rectangle (5,60 170x30), "State"
    Rectangle (5,90 170x30), "Substate"
    Rectangle (180,120 335x30), "%s", text variable: m_Instance.stat.sStatus
    Rectangle (180,150 335x30), "%s", tooltip "Additional information mostly used for description of errors", text variable: m_Instance.stat.sErrorText
    Rectangle (5,120 170x30), "Status"
    Rectangle (5,150 170x30), "Status Description"
    Rectangle (180,180 335x30), "%s", text variable: m_Instance.stat.sActionDesc
    Rectangle (180,210 335x30), "%s", text variable: m_Instance.stat.sEventDesc
    Rectangle (5,180 170x30), "Action"
    Rectangle (5,210 170x30), "Event"
    Rectangle (227,12 232x35), "%s", text variable: m_Instance.sName
    Checkbox (494,20 116x30), "Local Control", variable: m_Instance.stat.bLocal
    Rectangle (595,55 92x30), "Status"
    Rectangle (515,120 30x30), "%d", text variable: m_Instance.stat.nStatus
    Rectangle (739,55 92x30), "Switches"
    Button (350,450 150x30), "MOVE VEL-", input disabled if: NOT m_Instance.stat.bLocal OR NOT m_Instance.in_bSafe
        OnMouseDown: execute {
            m_Instance.ctrl.bLocalCmd := TRUE;
            m_Instance.ctrl.nCommand := E_MOTOR_COMMAND.MOTOR_MOVE;
            m_Instance.ctrl.nMoveType := E_MOTOR_MOVE_TYPE.VELOCITY;
            m_Instance.ctrl.nDirection := MC_Negative_Direction;
            m_Instance.ctrl.bExecute := TRUE;
        }
    Button (190,450 150x30), "MOVE REL", input disabled if: NOT m_Instance.stat.bLocal OR NOT m_Instance.in_bSafe
        OnMouseDown: execute {
            m_Instance.ctrl.bLocalCmd := TRUE;
            m_Instance.ctrl.lrVelocity:=(m_Instance.cfg.lrDefaultVelocity);
            m_Instance.ctrl.nCommand := E_MOTOR_COMMAND.MOTOR_MOVE;
            m_Instance.ctrl.nMoveType := E_MOTOR_MOVE_TYPE.RELATIVE;
            m_Instance.ctrl.bExecute := TRUE;
        }
    Button (190,490 150x30), "SET POS", input disabled if: NOT m_Instance.stat.bLocal OR NOT m_Instance.in_bSafe
        OnMouseDown: execute {
            m_Instance.ctrl.bLocalCmd := TRUE;
            m_Instance.ctrl.nCommand := E_MOTOR_COMMAND.SET_POSITION;
            m_Instance.ctrl.bExecute := TRUE;
        }
    Rectangle (785,95 50x15), "USTOP"
    Ellipse (760,95 15x15), colour toggle: m_Instance.stat.signals[5].bActive
    Ellipse (760,115 15x15), colour toggle: m_Instance.stat.signals[4].bActive
    Ellipse (760,175 15x15), colour toggle: m_Instance.stat.signals[1].bActive
    Ellipse (760,194 15x15), colour toggle: m_Instance.stat.signals[0].bActive
    Ellipse (760,155 15x15), colour toggle: m_Instance.stat.signals[2].bActive
    Rectangle (785,134 50x15), "INDEX"
    Rectangle (785,115 50x15), "UHW"
    Rectangle (785,155 50x15), "REF"
    Rectangle (785,175 50x15), "LHW"
    Rectangle (785,194 50x15), "LSTOP"
    Ellipse (760,134 15x15), colour toggle: m_Instance.stat.signals[3].bActive
    Rectangle (545,290 95x20), "Speed (Pos)"
    Rectangle (750,345 105x25), "%.2f", text variable: m_Instance.stat.lrPosActual, input disabled if: false
    Rectangle (672,260 190x20), "Target Actual"
    Rectangle (545,348 95x20), "Position (ABS)"
    Rectangle (750,290 105x50), "%.2f", text variable: m_Instance.stat.lrVelActual, input disabled if: false
    Rectangle (645,315 105x25), "%.2f", text variable: m_Instance.ctrl.lrVelocity
        OnMouseDown: write the text variable via Default
    Rectangle (545,403 95x20), "Backlash"
    Rectangle (645,400 105x25), "%.2f", text variable: m_Instance.cfg.lrBacklash
        OnMouseDown: write the text variable via Default
    Rectangle (545,315 95x25), "Speed (Vel)"
    Rectangle (645,345 105x25), "%.2f", tooltip "Absolute position used by "MOVE ABS"", text variable: m_Instance.ctrl.lrPosition
        OnMouseDown: write the text variable via Default
    Rectangle (645,290 105x25), "%.2f", text variable: m_Instance.cfg.lrDefaultVelocity
        OnMouseDown: write the text variable via Default
    Rectangle (605,171 90x25), "Brake Active"
    Ellipse (580,175 15x15), tooltip "RED = Applied BLANK = Released", colour toggle: (m_Instance.stat.bBrakeActive) <> 0
    Ellipse (580,95 15x15), tooltip "GREEN = Initialised RED = Not Initialised", text variable: m_Instance.stat.bInitialised, colour toggle: m_Instance.stat.bInitialised
    Rectangle (605,91 90x25), "Initialised"
    Rectangle (605,111 125x25), "Controller Enabled"
    Rectangle (605,131 90x24), "Axis Ready"
    Rectangle (605,151 90x25), "Brake Used"
    Ellipse (580,115 15x15), tooltip "GREEN = Enabled RED = Disabled", colour toggle: m_Instance.stat.bEnabled
    Ellipse (580,135 15x15), tooltip "GREEN = Ready RED = Not Ready", colour toggle: m_Instance.stat.bAxisReady
    Ellipse (580,155 15x15), tooltip "BLUE = Used BLANK = Not Used", colour toggle: m_Instance.cfg.bUseBrake
    Rectangle (578,230 20x20), "%d", text variable: m_Instance.stat.nInitStep
    Rectangle (605,228 90x25), "INIT Step"
    Rectangle (5,240 170x30), "RPC Call Status"
    Rectangle (180,240 335x30), "%s", text variable: m_Instance.stat.sRPCErrorText
    Rectangle (605,191 90x25), "In Position"
    Ellipse (580,195 15x15), tooltip "GREEN = In Position BLANK = Not In Position (or not used)", colour toggle: (m_Instance.stat.bInPosition) <> 0
    Button (645,435 105x50), "ENABLE AXIS", input disabled if: NOT m_Instance.stat.bLocal OR NOT m_Instance.in_bSafe
        OnMouseDown: execute { m_Instance.stat.bEnabled := TRUE; }
    Button (752,435 105x50), "DISABLE AXIS", input disabled if: NOT m_Instance.stat.bLocal OR NOT m_Instance.in_bSafe
        OnMouseDown: execute { m_Instance.stat.bEnabled := FALSE; }
    Rectangle (620,15 203x30), "User Units: '%s'", text variable: m_Instance.stat.axis.sUnits
    Rectangle (5,10 99x30), "Ver: %s", tooltip "'Motor.library version'", text variable: m_Instance.stat.sLibVersion, input disabled if: true
    Rectangle (545,373 95x20), "Offset (REL)"
    Rectangle (645,370 105x25), "%.2f", tooltip "Relative offset used by "MOVE REL"", text variable: m_Instance.ctrl.lrOffset
        OnMouseDown: write the text variable via Default
    Lamp1 (552,436 50x50), tooltip "If active, it is not safe to operate the motor.", variable: NOT m_Instance.in_bSafe, invisible if: m_Instance.in_bSafe, style: Lamp-Lamp1-Red
    Rectangle (526,491 100x30), "Unsafe!", invisible if: m_Instance.in_bSafe
END_VISUALIZATION

// ---- VISUs/Tracking/GUI_ADC_Motor1.TcVIS
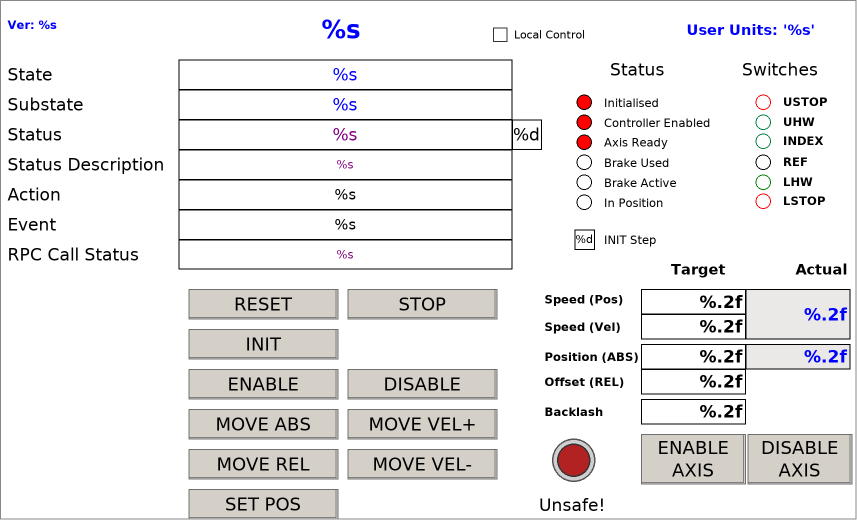
VISUALIZATION GUI_ADC_Motor1  // 857x520
    Frame (0,0 857x520)
        shows GUI_TEMPLATE_MOTOR_CONTROL(m_Instance := MAIN.adc.motor1)
END_VISUALIZATION

// ---- VISUs/Tracking/GUI_ADC_Motor2.TcVIS
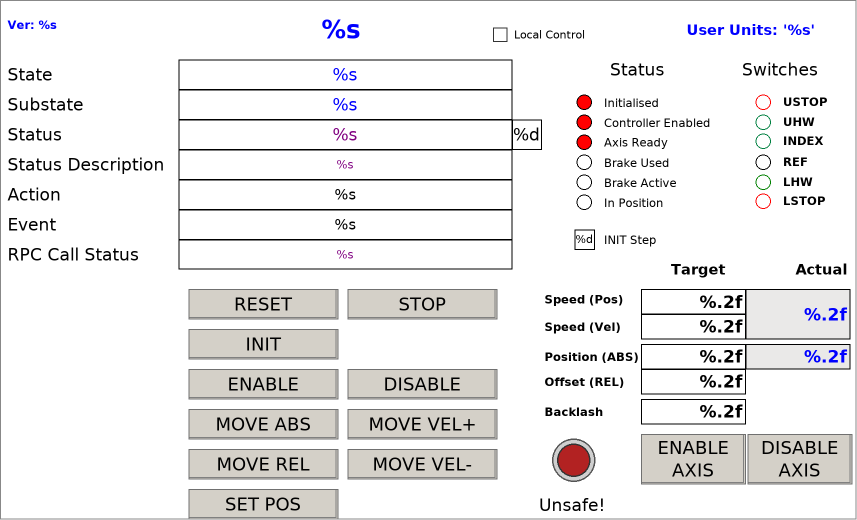
VISUALIZATION GUI_ADC_Motor2  // 857x520
    Frame (0,0 857x520)
        shows GUI_TEMPLATE_MOTOR_CONTROL(m_Instance := MAIN.adc.motor2)
END_VISUALIZATION

// ---- VISUs/Tracking/GUI_MA_ADC.TcVIS
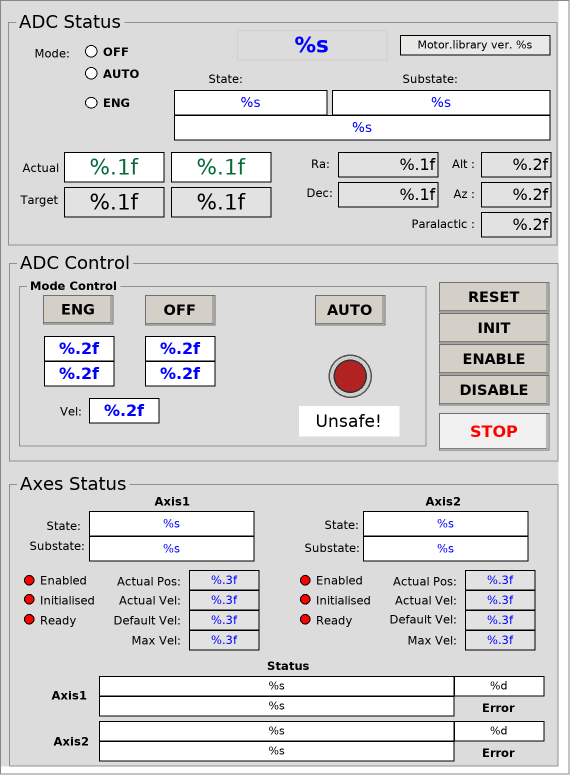
VISUALIZATION GUI_MA_ADC  // 570x775
    Frame (0,0 568x773)
        shows GUI_TEMPLATE_MA_ADC(m_DeviceName := 'ADC', m_Instance := MAIN.adc)
END_VISUALIZATION

// ---- VISUs/Tracking/GUI_MA_DROT.TcVIS
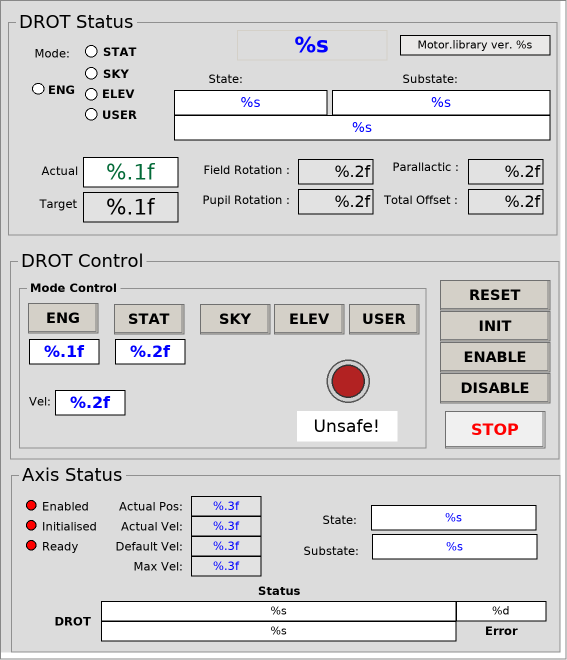
VISUALIZATION GUI_MA_DROT  // 567x660
    Frame (0,0 565x658)
        shows GUI_TEMPLATE_MA_DROT(m_DeviceName := 'DROT', m_Instance := MAIN.drot)
END_VISUALIZATION

// ---- VISUs/Tracking/GUI_DROT_Cfg.TcVIS
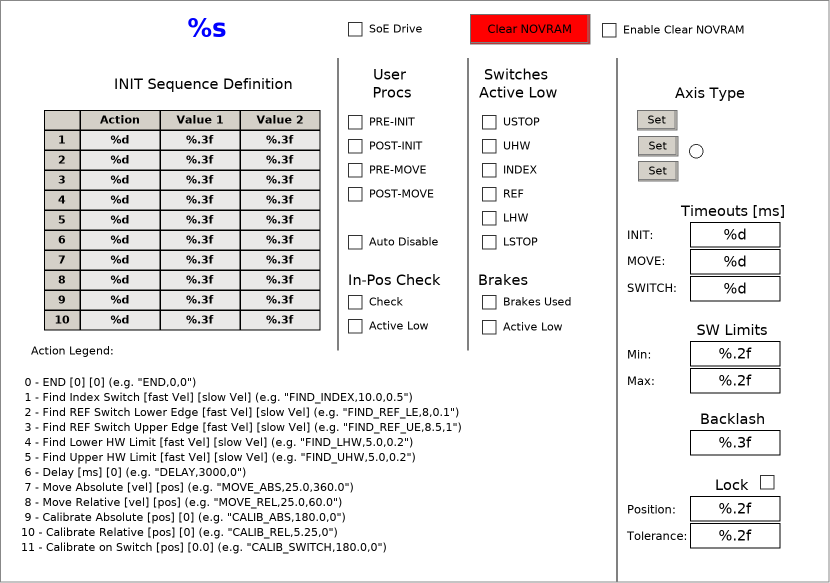
VISUALIZATION GUI_DROT_Cfg  // 830x583
    Frame (0,0 828x581)
        shows GUI_TEMPLATE_MOTOR_CONFIG(m_Instance := MAIN.drot.motor)
END_VISUALIZATION

// ---- VISUs/Tracking/GUI_DROT_Motor.TcVIS
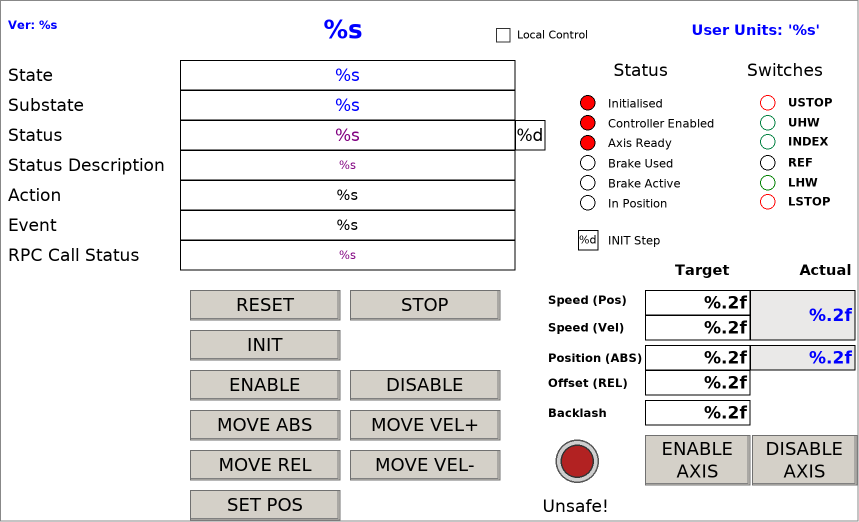
VISUALIZATION GUI_DROT_Motor  // 859x522
    Frame (0,0 857x520)
        shows GUI_TEMPLATE_MOTOR_CONTROL(m_Instance := MAIN.drot.motor)
END_VISUALIZATION

// ---- VISUs/Tracking/GUI_TIMER.TcVIS
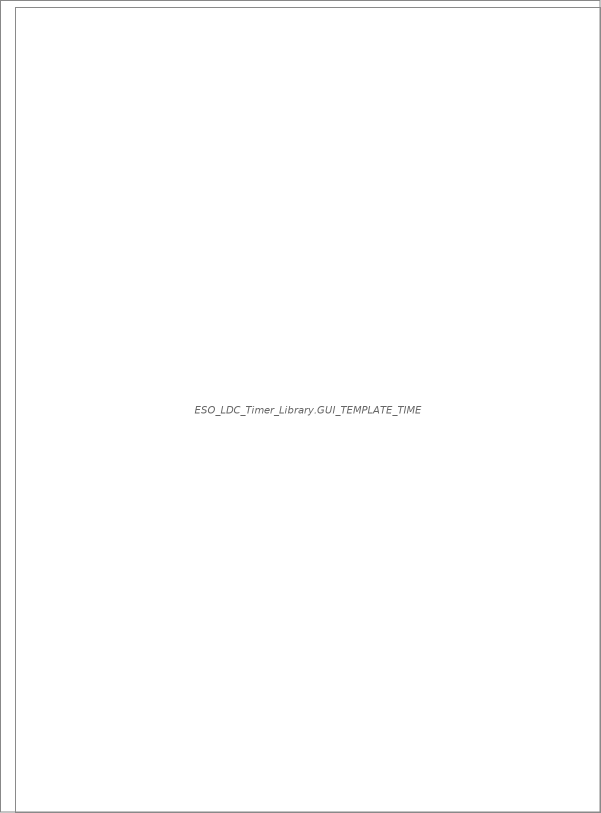
VISUALIZATION GUI_TIMER  // 601x813
    Frame (15,7 586x806)
        shows ESO_LDC_Timer_Library.GUI_TEMPLATE_TIME(m_DeviceName := 'MAIN.fbTimer', m_Instance := MAIN.time_data)
END_VISUALIZATION
